KUKA KRL program: MyProgram_173().src

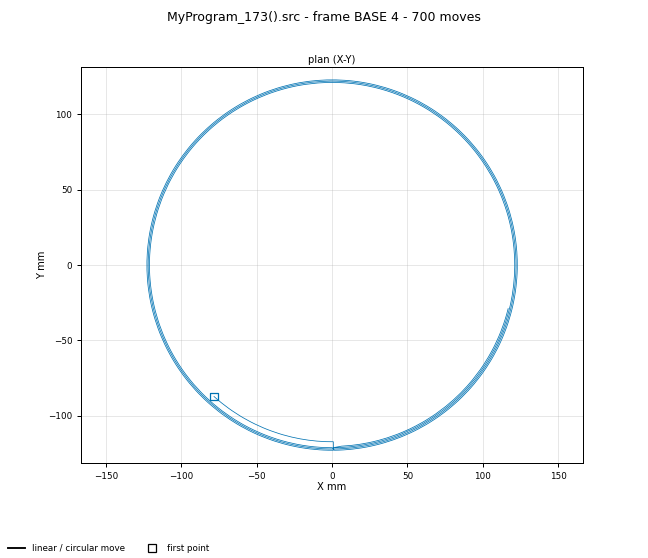
[picture p0: tool path of MyProgram_173().src in frame BASE 4, 700 of 700 moves have a stored position in this frame; points joined in program order, loops and branches not executed]
&ACCESS RVP
&REL 1
&PARAM TEMPLATE = C:\KRC\Roboter\Template\vorgabe
&PARAM EDITMASK = *
DEF MyProgram_173()
; ---- Setting reference (Base) ----
$BASE = BASE_DATA[4]

; --------------------------
; ---- Setting tool (TCP) ----
$TOOL = TOOL_DATA[3]
; --------------------------

$VEL.CP = VEL_APROX_PRINT
Startdeposition()
$VEL.CP = VEL_PRINT
LIN {X -78.3175,Y -87.2157,Z 128,A -135.2018,B 24.9548,C -1.5536,E1 24.894,E2 221.2459} C_DIS
LIN {X -76.0204,Y -89.2249,Z 128,A -133.7214,B 24.955,C -1.5502,E1 24.8972,E2 219.7678} C_DIS
LIN {X -73.3158,Y -91.4624,Z 128,A -132.0203,B 24.9552,C -1.5463,E1 24.9008,E2 218.0696} C_DIS
LIN {X -70.7779,Y -93.4392,Z 128,A -130.557,B 24.9556,C -1.5388,E1 24.904,E2 216.6188} C_DIS
LIN {X -68.6874,Y -94.988,Z 128,A -129.0705,B 24.9552,C -1.5458,E1 24.9074,E2 215.1104} C_DIS
LIN {X -66.3132,Y -96.6605,Z 128,A -127.7459,B 24.9556,C -1.5393,E1 24.9105,E2 213.7967} C_DIS
LIN {X -63.7074,Y -98.3959,Z 128,A -126.2103,B 24.9557,C -1.5371,E1 24.914,E2 212.2613} C_DIS
LIN {X -61.2786,Y -99.9267,Z 128,A -124.8024,B 24.9558,C -1.5352,E1 24.9174,E2 210.8536} C_DIS
LIN {X -58.8133,Y -101.3972,Z 128,A -123.3955,B 24.956,C -1.5333,E1 24.9208,E2 209.447} C_DIS
LIN {X -56.1243,Y -102.9093,Z 128,A -122.0747,B 24.9565,C -1.5231,E1 24.9239,E2 208.1466} C_DIS
LIN {X -53.9775,Y -104.0535,Z 128,A -120.6902,B 24.9561,C -1.53,E1 24.9274,E2 206.7418} C_DIS
LIN {X -51.181,Y -105.4557,Z 128,A -119.157,B 24.9562,C -1.5283,E1 24.9312,E2 205.2087} C_DIS
LIN {X -48.3648,Y -106.7758,Z 128,A -117.8498,B 24.9569,C -1.5172,E1 24.9345,E2 203.9245} C_DIS
LIN {X -45.8347,Y -107.8864,Z 128,A -116.3218,B 24.9565,C -1.5235,E1 24.9385,E2 202.378} C_DIS
LIN {X -43.5316,Y -108.8379,Z 128,A -114.9638,B 24.9562,C -1.5284,E1 24.942,E2 201.0053} C_DIS
LIN {X -40.5891,Y -109.9678,Z 128,A -113.5212,B 24.9566,C -1.5227,E1 24.9458,E2 199.5733} C_DIS
LIN {X -37.8192,Y -110.9506,Z 128,A -112.1239,B 24.9567,C -1.5197,E1 24.9494,E2 198.1804} C_DIS
LIN {X -35.2434,Y -111.7962,Z 128,A -110.8198,B 24.9568,C -1.5177,E1 24.9529,E2 196.8786} C_DIS
LIN {X -32.6052,Y -112.5946,Z 128,A -109.2722,B 24.9564,C -1.5257,E1 24.9571,E2 195.3097} C_DIS
LIN {X -29.336,Y -113.4884,Z 128,A -107.7138,B 24.9567,C -1.5203,E1 24.9613,E2 193.7616} C_DIS
LIN {X -26.8263,Y -114.1085,Z 128,A -106.5879,B 24.9571,C -1.5135,E1 24.9643,E2 192.6504} C_DIS
LIN {X -24.0235,Y -114.7313,Z 128,A -105.0697,B 24.9568,C -1.518,E1 24.9685,E2 191.1197} C_DIS
LIN {X -21.2072,Y -115.2851,Z 128,A -103.6628,B 24.9568,C -1.5176,E1 24.9723,E2 189.7121} C_DIS
LIN {X -18.6199,Y -115.7324,Z 128,A -102.2849,B 24.9566,C -1.5214,E1 24.9762,E2 188.3239} C_DIS
LIN {X -15.7808,Y -116.1536,Z 128,A -100.8781,B 24.9566,C -1.5213,E1 24.98,E2 186.9163} C_DIS
LIN {X -12.6612,Y -116.5336,Z 128,A -99.4416,B 24.9569,C -1.5166,E1 24.984,E2 185.49} C_DIS
LIN {X -10.0626,Y -116.788,Z 128,A -98.1635,B 24.9569,C -1.5166,E1 24.9876,E2 184.2113} C_DIS
LIN {X -6.9466,Y -117.0135,Z 128,A -96.6383,B 24.9569,C -1.5166,E1 24.9918,E2 182.6857} C_DIS
LIN {X -4.0837,Y -117.1484,Z 128,A -95.3376,B 24.9572,C -1.5121,E1 24.9954,E2 181.3951} C_DIS
LIN {X -1.1778,Y -117.2135,Z 128,A -93.9306,B 24.9572,C -1.5118,E1 24.9993,E2 179.9889} C_DIS
LIN {X 0.813,Y -117.2142,Z 128,A -93.1077,B 24.9576,C -1.5052,E1 25.0016,E2 179.1816} C_DIS
Enddeposition()
LIN {X 0.8728,Y -122.8508,Z 129,A -93.006,B 24.9623,C -1.4183,E1 25.0013,E2 179.2858} C_DIS
Startdeposition()
$VEL.CP = VEL_PRINT
LIN {X -2.5785,Y -122.8272,Z 129,A -94.9222,B 24.9631,C -1.4034,E1 24.9959,E2 181.2373} C_DIS
LIN {X -5.5921,Y -122.7269,Z 129,A -96.2871,B 24.9631,C -1.4052,E1 24.9921,E2 182.5982} C_DIS
LIN {X -8.6023,Y -122.5527,Z 129,A -97.6934,B 24.9631,C -1.4052,E1 24.9881,E2 184.0051} C_DIS
LIN {X -12.042,Y -122.2646,Z 129,A -99.303,B 24.9631,C -1.4052,E1 24.9837,E2 185.6154} C_DIS
LIN {X -14.6053,Y -121.983,Z 129,A -100.5473,B 24.9631,C -1.4035,E1 24.9802,E2 186.8646} C_DIS
LIN {X -17.5945,Y -121.5879,Z 129,A -101.9132,B 24.963,C -1.4057,E1 24.9764,E2 188.2263} C_DIS
LIN {X -20.5731,Y -121.1195,Z 129,A -103.3204,B 24.963,C -1.4061,E1 24.9725,E2 189.634} C_DIS
LIN {X -23.5393,Y -120.5781,Z 129,A -104.7183,B 24.963,C -1.407,E1 24.9687,E2 191.0311} C_DIS
LIN {X -26.9179,Y -119.871,Z 129,A -106.339,B 24.963,C -1.4072,E1 24.9643,E2 192.6533} C_DIS
LIN {X -29.8516,Y -119.1743,Z 129,A -107.7472,B 24.9629,C -1.4079,E1 24.9605,E2 194.0619} C_DIS
LIN {X -32.7673,Y -118.4058,Z 129,A -109.155,B 24.9629,C -1.4087,E1 24.9567,E2 195.4699} C_DIS
LIN {X -35.6633,Y -117.566,Z 129,A -110.5633,B 24.9628,C -1.4096,E1 24.9529,E2 196.8785} C_DIS
LIN {X -38.1224,Y -116.7898,Z 129,A -111.7683,B 24.9628,C -1.4104,E1 24.9497,E2 198.0836} C_DIS
LIN {X -41.389,Y -115.6745,Z 129,A -113.3811,B 24.9627,C -1.4117,E1 24.9454,E2 199.6966} C_DIS
LIN {X -44.0204,Y -114.6977,Z 129,A -114.7031,B 24.9627,C -1.4123,E1 24.942,E2 201.0198} C_DIS
LIN {X -46.6107,Y -113.6689,Z 129,A -116.0365,B 24.9627,C -1.4121,E1 24.9385,E2 202.3567} C_DIS
LIN {X -49.3862,Y -112.4908,Z 129,A -117.4048,B 24.9625,C -1.4154,E1 24.935,E2 203.7205} C_DIS
LIN {X -52.5278,Y -111.0607,Z 129,A -119.0187,B 24.9624,C -1.417,E1 24.9309,E2 205.3344} C_DIS
LIN {X -55.2375,Y -109.7381,Z 129,A -120.4286,B 24.9624,C -1.4186,E1 24.9274,E2 206.7443} C_DIS
LIN {X -57.914,Y -108.3495,Z 129,A -121.8387,B 24.9622,C -1.4203,E1 24.9239,E2 208.1543} C_DIS
LIN {X -60.1744,Y -107.1084,Z 129,A -123.0452,B 24.9622,C -1.4218,E1 24.921,E2 209.3606} C_DIS
LIN {X -63.1607,Y -105.3773,Z 129,A -124.6598,B 24.962,C -1.4239,E1 24.9171,E2 210.9751} C_DIS
LIN {X -65.7278,Y -103.7955,Z 129,A -126.0709,B 24.962,C -1.4259,E1 24.9137,E2 212.386} C_DIS
LIN {X -67.8803,Y -102.3984,Z 129,A -127.3153,B 24.962,C -1.4256,E1 24.9108,E2 213.635} C_DIS
LIN {X -70.7416,Y -100.4453,Z 129,A -128.8932,B 24.9617,C -1.43,E1 24.9072,E2 215.2078} C_DIS
LIN {X -72.8331,Y -98.9369,Z 129,A -130.1005,B 24.9616,C -1.4319,E1 24.9045,E2 216.4148} C_DIS
LIN {X -75.2392,Y -97.1197,Z 129,A -131.5534,B 24.9616,C -1.4324,E1 24.9013,E2 217.8719} C_DIS
LIN {X -77.9391,Y -94.9691,Z 129,A -133.1283,B 24.9613,C -1.4369,E1 24.8979,E2 219.4419} C_DIS
LIN {X -79.914,Y -93.3109,Z 129,A -134.336,B 24.9613,C -1.4391,E1 24.8953,E2 220.6492} C_DIS
LIN {X -82.1799,Y -91.3216,Z 129,A -135.7483,B 24.9611,C -1.4416,E1 24.8923,E2 222.061} C_DIS
LIN {X -84.7143,Y -88.9782,Z 129,A -137.3655,B 24.9609,C -1.4446,E1 24.889,E2 223.6778} C_DIS
LIN {X -86.8724,Y -86.8724,Z 129,A -138.7777,B 24.9608,C -1.4473,E1 24.8862,E2 225.0895} C_DIS
LIN {X -88.6753,Y -85.0287,Z 129,A -139.9861,B 24.9606,C -1.4498,E1 24.8839,E2 226.2973} C_DIS
LIN {X -90.7691,Y -82.79,Z 129,A -141.4561,B 24.9606,C -1.4512,E1 24.8811,E2 227.7704} C_DIS
LIN {X -93.0278,Y -80.2463,Z 129,A -143.017,B 24.9603,C -1.4559,E1 24.8782,E2 229.3269} C_DIS
LIN {X -94.6901,Y -78.2749,Z 129,A -144.2259,B 24.9601,C -1.4585,E1 24.8761,E2 230.5353} C_DIS
LIN {X -96.5825,Y -75.9275,Z 129,A -145.6807,B 24.9601,C -1.4598,E1 24.8735,E2 231.994} C_DIS
LIN {X -98.679,Y -73.1853,Z 129,A -147.2578,B 24.9598,C -1.4652,E1 24.8709,E2 233.5657} C_DIS
LIN {X -100.4453,Y -70.7416,Z 129,A -148.6716,B 24.9596,C -1.4684,E1 24.8686,E2 234.9787} C_DIS
LIN {X -101.9064,Y -68.6167,Z 129,A -149.881,B 24.9594,C -1.4712,E1 24.8667,E2 236.1874} C_DIS
LIN {X -103.5597,Y -66.0952,Z 129,A -151.2749,B 24.9592,C -1.4755,E1 24.8646,E2 237.5782} C_DIS
LIN {X -105.1505,Y -63.5338,Z 129,A -152.7094,B 24.9591,C -1.478,E1 24.8625,E2 239.0141} C_DIS
LIN {X -106.8956,Y -60.5556,Z 129,A -154.3286,B 24.9589,C -1.4819,E1 24.8602,E2 240.6324} C_DIS
LIN {X -108.3495,Y -57.914,Z 129,A -155.7433,B 24.9587,C -1.4854,E1 24.8583,E2 242.0461} C_DIS
LIN {X -109.5394,Y -55.6263,Z 129,A -156.9533,B 24.9585,C -1.4885,E1 24.8568,E2 243.2553} C_DIS
LIN {X -111.0607,Y -52.5278,Z 129,A -158.5729,B 24.9583,C -1.4927,E1 24.8548,E2 244.8738} C_DIS
LIN {X -112.3163,Y -49.7864,Z 129,A -159.9877,B 24.9581,C -1.4963,E1 24.8532,E2 246.2876} C_DIS
LIN {X -113.3348,Y -47.4173,Z 129,A -161.2395,B 24.958,C -1.4977,E1 24.8519,E2 247.543} C_DIS
LIN {X -114.4643,Y -44.6217,Z 129,A -162.6133,B 24.9577,C -1.5033,E1 24.8504,E2 248.9112} C_DIS
LIN {X -115.5249,Y -41.7991,Z 129,A -164.0285,B 24.9574,C -1.5071,E1 24.8491,E2 250.3253} C_DIS
LIN {X -116.6554,Y -38.5377,Z 129,A -165.6487,B 24.9572,C -1.5115,E1 24.8476,E2 251.9443} C_DIS
LIN {X -117.4367,Y -36.0803,Z 129,A -166.8595,B 24.957,C -1.5149,E1 24.8466,E2 253.154} C_DIS
LIN {X -118.2868,Y -33.1874,Z 129,A -168.275,B 24.9568,C -1.5188,E1 24.8455,E2 254.5683} C_DIS
LIN {X -119.0657,Y -30.2745,Z 129,A -169.6906,B 24.9566,C -1.5228,E1 24.8445,E2 255.9828} C_DIS
LIN {X -119.801,Y -27.2211,Z 129,A -171.1534,B 24.9563,C -1.5274,E1 24.8436,E2 257.443} C_DIS
LIN {X -120.4955,Y -23.9681,Z 129,A -172.727,B 24.9561,C -1.5313,E1 24.8427,E2 259.0166} C_DIS
LIN {X -121.0193,Y -21.1602,Z 129,A -174.0531,B 24.9558,C -1.5358,E1 24.842,E2 260.3399} C_DIS
LIN {X -121.5265,Y -18.0267,Z 129,A -175.5587,B 24.9556,C -1.5395,E1 24.8414,E2 261.8458} C_DIS
LIN {X -121.8761,Y -15.4719,Z 129,A -176.8112,B 24.9555,C -1.5412,E1 24.8409,E2 263.1016} C_DIS
LIN {X -122.2191,Y -12.4762,Z 129,A -178.1858,B 24.9552,C -1.5471,E1 24.8405,E2 264.4704} C_DIS
LIN {X -122.5233,Y -9.0379,Z 129,A -179.807,B 24.9549,C -1.5518,E1 24.8402,E2 266.0901} C_DIS
LIN {X -122.7082,Y -6.0283,Z 129,A 178.7771,B 24.9546,C -1.5559,E1 24.8399,E2 267.5046} C_DIS
LIN {X -122.8058,Y -3.4514,Z 129,A 177.5245,B 24.9546,C -1.5577,E1 24.8399,E2 268.7605} C_DIS
LIN {X -122.8542,Y -0.3629,Z 129,A 176.0949,B 24.9542,C -1.5629,E1 24.8398,E2 270.1864} C_DIS
LIN {X -122.8272,Y 2.5785,Z 129,A 174.6923,B 24.954,C -1.5661,E1 24.8398,E2 271.5899} C_DIS
LIN {X -122.7269,Y 5.5921,Z 129,A 173.3176,B 24.9537,C -1.572,E1 24.84,E2 272.9587} C_DIS
LIN {X -122.5604,Y 8.4883,Z 129,A 171.9386,B 24.9535,C -1.5753,E1 24.8402,E2 274.3381} C_DIS
LIN {X -122.2646,Y 12.042,Z 129,A 170.2806,B 24.9532,C -1.581,E1 24.8407,E2 275.9927} C_DIS
LIN {X -121.9322,Y 15.0389,Z 129,A 168.8642,B 24.9529,C -1.5851,E1 24.8411,E2 277.4076} C_DIS
LIN {X -121.5879,Y 17.5945,Z 129,A 167.6531,B 24.9527,C -1.5887,E1 24.8416,E2 278.6174} C_DIS
LIN {X -121.0475,Y 21.0037,Z 129,A 166.0319,B 24.9524,C -1.5934,E1 24.8423,E2 280.237} C_DIS
LIN {X -120.4955,Y 23.9681,Z 129,A 164.616,B 24.9522,C -1.5976,E1 24.8431,E2 281.6513} C_DIS
LIN {X -119.871,Y 26.9179,Z 129,A 163.2,B 24.9519,C -1.6017,E1 24.8439,E2 283.0658} C_DIS
LIN {X -119.1743,Y 29.8516,Z 129,A 161.7838,B 24.9517,C -1.6058,E1 24.8448,E2 284.4805} C_DIS
LIN {X -118.4058,Y 32.7673,Z 129,A 160.368,B 24.9514,C -1.6099,E1 24.8459,E2 285.8947} C_DIS
LIN {X -117.566,Y 35.6633,Z 129,A 158.9522,B 24.9512,C -1.614,E1 24.847,E2 287.3091} C_DIS
LIN {X -116.6554,Y 38.5377,Z 129,A 157.5361,B 24.9509,C -1.618,E1 24.8482,E2 288.7237} C_DIS
LIN {X -115.8191,Y 40.977,Z 129,A 156.3254,B 24.9507,C -1.6215,E1 24.8493,E2 289.9329} C_DIS
LIN {X -114.7786,Y 43.807,Z 129,A 154.8682,B 24.9506,C -1.6237,E1 24.8507,E2 291.3931} C_DIS
LIN {X -113.6689,Y 46.6107,Z 129,A 153.4526,B 24.9504,C -1.6277,E1 24.8522,E2 292.8072} C_DIS
LIN {X -112.4908,Y 49.3862,Z 129,A 152.0784,B 24.95,C -1.6334,E1 24.8537,E2 294.1753} C_DIS
LIN {X -111.0607,Y 52.5278,Z 129,A 150.4581,B 24.9497,C -1.6378,E1 24.8556,E2 295.794} C_DIS
LIN {X -109.932,Y 54.8464,Z 129,A 149.2062,B 24.9497,C -1.6393,E1 24.8572,E2 297.0489} C_DIS
LIN {X -108.3495,Y 57.914,Z 129,A 147.6276,B 24.9493,C -1.6455,E1 24.8592,E2 298.6213} C_DIS
LIN {X -107.1084,Y 60.1744,Z 129,A 146.3944,B 24.9491,C -1.6477,E1 24.8609,E2 299.8556} C_DIS
LIN {X -105.3773,Y 63.1607,Z 129,A 144.7972,B 24.9488,C -1.6529,E1 24.8632,E2 301.4487} C_DIS
LIN {X -103.7955,Y 65.7278,Z 129,A 143.3822,B 24.9486,C -1.6566,E1 24.8652,E2 302.8621} C_DIS
LIN {X -102.1512,Y 68.2552,Z 129,A 141.9675,B 24.9483,C -1.6602,E1 24.8674,E2 304.2753} C_DIS
LIN {X -100.4454,Y 70.7416,Z 129,A 140.5528,B 24.9481,C -1.6638,E1 24.8697,E2 305.6885} C_DIS
LIN {X -98.9369,Y 72.8331,Z 129,A 139.3428,B 24.9479,C -1.6668,E1 24.8717,E2 306.8971} C_DIS
LIN {X -97.1197,Y 75.2392,Z 129,A 137.9283,B 24.9477,C -1.6703,E1 24.8741,E2 308.3102} C_DIS
LIN {X -95.2749,Y 77.5618,Z 129,A 136.5307,B 24.9475,C -1.6734,E1 24.8765,E2 309.7069} C_DIS
LIN {X -93.3109,Y 79.914,Z 129,A 135.0585,B 24.9475,C -1.6752,E1 24.8792,E2 311.1814} C_DIS
LIN {X -91.0304,Y 82.5052,Z 129,A 133.4814,B 24.9471,C -1.6808,E1 24.8821,E2 312.7524} C_DIS
LIN {X -88.9782,Y 84.7143,Z 129,A 132.0672,B 24.9469,C -1.684,E1 24.8848,E2 314.1652} C_DIS
LIN {X -86.8724,Y 86.8724,Z 129,A 130.6539,B 24.9467,C -1.6871,E1 24.8875,E2 315.577} C_DIS
LIN {X -84.7143,Y 88.9782,Z 129,A 129.2402,B 24.9465,C -1.6902,E1 24.8904,E2 316.9893} C_DIS
LIN {X -82.6505,Y 90.8971,Z 129,A 127.9097,B 24.9463,C -1.6926,E1 24.8931,E2 318.3195} C_DIS
LIN {X -80.5751,Y 92.7406,Z 129,A 126.6269,B 24.9461,C -1.6961,E1 24.8958,E2 319.5989} C_DIS
LIN {X -78.2749,Y 94.6901,Z 129,A 125.2051,B 24.9459,C -1.6986,E1 24.8988,E2 321.0203} C_DIS
LIN {X -75.9275,Y 96.5825,Z 129,A 123.7923,B 24.9458,C -1.7014,E1 24.9019,E2 322.4317} C_DIS
LIN {X -73.5344,Y 98.4168,Z 129,A 122.3381,B 24.9457,C -1.7022,E1 24.9052,E2 323.8891} C_DIS
LIN {X -71.1398,Y 100.1613,Z 129,A 120.9848,B 24.9454,C -1.7064,E1 24.9082,E2 325.2373} C_DIS
LIN {X -68.6167,Y 101.9064,Z 129,A 119.5548,B 24.9452,C -1.7093,E1 24.9115,E2 326.6652} C_DIS
LIN {X -66.0952,Y 103.5597,Z 129,A 118.1429,B 24.9451,C -1.7117,E1 24.9148,E2 328.0758} C_DIS
LIN {X -63.5338,Y 105.1505,Z 129,A 116.7309,B 24.9449,C -1.7141,E1 24.9182,E2 329.4866} C_DIS
LIN {X -60.5556,Y 106.8956,Z 129,A 115.1146,B 24.9448,C -1.7167,E1 24.9221,E2 331.1015} C_DIS
LIN {X -57.914,Y 108.3495,Z 129,A 113.7034,B 24.9446,C -1.7189,E1 24.9256,E2 332.5115} C_DIS
LIN {X -55.4274,Y 109.6411,Z 129,A 112.4075,B 24.9445,C -1.7216,E1 24.9288,E2 333.8045} C_DIS
LIN {X -52.5278,Y 111.0607,Z 129,A 110.881,B 24.9444,C -1.723,E1 24.9326,E2 335.3314} C_DIS
LIN {X -49.7864,Y 112.3163,Z 129,A 109.4703,B 24.9442,C -1.725,E1 24.9362,E2 336.741} C_DIS
LIN {X -47.4173,Y 113.3348,Z 129,A 108.2224,B 24.9442,C -1.7247,E1 24.9394,E2 337.9923} C_DIS
LIN {X -44.6217,Y 114.4643,Z 129,A 106.8532,B 24.944,C -1.7283,E1 24.943,E2 339.3559} C_DIS
LIN {X -41.7991,Y 115.5249,Z 129,A 105.4431,B 24.944,C -1.73,E1 24.9466,E2 340.765} C_DIS
LIN {X -38.5377,Y 116.6554,Z 129,A 103.8291,B 24.9438,C -1.7318,E1 24.9509,E2 342.3778} C_DIS
LIN {X -36.0803,Y 117.4367,Z 129,A 102.6232,B 24.9438,C -1.7331,E1 24.9541,E2 343.5827} C_DIS
LIN {X -33.1874,Y 118.2868,Z 129,A 101.1725,B 24.9438,C -1.7326,E1 24.958,E2 345.037} C_DIS
LIN {X -29.8516,Y 119.1743,Z 129,A 99.6006,B 24.9435,C -1.7359,E1 24.9623,E2 346.6034} C_DIS
LIN {X -27.296,Y 119.7837,Z 129,A 98.378,B 24.9435,C -1.7372,E1 24.9656,E2 347.8245} C_DIS
LIN {X -23.9681,Y 120.4955,Z 129,A 96.7827,B 24.9434,C -1.7381,E1 24.9699,E2 349.4194} C_DIS
LIN {X -21.0037,Y 121.0475,Z 129,A 95.3741,B 24.9434,C -1.7391,E1 24.9738,E2 350.8271} C_DIS
LIN {X -18.0267,Y 121.5265,Z 129,A 93.9659,B 24.9433,C -1.74,E1 24.9777,E2 352.2345} C_DIS
LIN {X -15.4719,Y 121.8761,Z 129,A 92.7616,B 24.9433,C -1.7407,E1 24.981,E2 353.438} C_DIS
LIN {X -12.042,Y 122.2646,Z 129,A 91.1499,B 24.9432,C -1.7415,E1 24.9855,E2 355.0489} C_DIS
LIN {X -9.4731,Y 122.4885,Z 129,A 89.9457,B 24.9432,C -1.742,E1 24.9888,E2 356.2523} C_DIS
LIN {X -6.0283,Y 122.7082,Z 129,A 88.3348,B 24.9431,C -1.7425,E1 24.9933,E2 357.8625} C_DIS
LIN {X -3.5053,Y 122.8041,Z 129,A 87.1059,B 24.9432,C -1.7405,E1 24.9968,E2 359.0963} C_DIS
LIN {X 0,Y 122.8562,Z 129,A 85.5207,B 24.9431,C -1.7432,E1 25.0012,E2 360.6753} C_DIS
LIN {X 2.5785,Y 122.8272,Z 129,A 84.2766,B 24.9431,C -1.7414,E1 25.0047,E2 361.9233} C_DIS
LIN {X 5.5921,Y 122.7269,Z 129,A 82.9112,B 24.9431,C -1.7434,E1 25.0085,E2 363.2836} C_DIS
LIN {X 8.5036,Y 122.5594,Z 129,A 81.5373,B 24.9431,C -1.7428,E1 25.0123,E2 364.6585} C_DIS
LIN {X 11.6073,Y 122.3047,Z 129,A 80.0581,B 24.9431,C -1.7414,E1 25.0164,E2 366.1401} C_DIS
LIN {X 14.6053,Y 121.983,Z 129,A 78.6935,B 24.9431,C -1.7431,E1 25.0202,E2 367.4998} C_DIS
LIN {X 17.5945,Y 121.5879,Z 129,A 77.247,B 24.9432,C -1.7408,E1 25.0242,E2 368.9503} C_DIS
LIN {X 20.5731,Y 121.1195,Z 129,A 75.8414,B 24.9432,C -1.7404,E1 25.0281,E2 370.3555} C_DIS
LIN {X 23.8641,Y 120.5155,Z 129,A 74.3206,B 24.9432,C -1.7416,E1 25.0322,E2 371.8717} C_DIS
LIN {X 26.9179,Y 119.871,Z 129,A 72.8697,B 24.9432,C -1.7411,E1 25.0362,E2 373.322} C_DIS
LIN {X 29.8516,Y 119.1743,Z 129,A 71.465,B 24.9432,C -1.7403,E1 25.04,E2 374.7265} C_DIS
LIN {X 32.7673,Y 118.4058,Z 129,A 70.0609,B 24.9432,C -1.7395,E1 25.0438,E2 376.1303} C_DIS
LIN {X 35.1793,Y 117.7096,Z 129,A 68.8387,B 24.9435,C -1.7362,E1 25.0471,E2 377.358} C_DIS
LIN {X 38.1224,Y 116.7898,Z 129,A 67.4561,B 24.9435,C -1.7377,E1 25.0507,E2 378.7347} C_DIS
LIN {X 40.977,Y 115.8191,Z 129,A 66.0524,B 24.9435,C -1.7366,E1 25.0544,E2 380.1382} C_DIS
LIN {X 43.8071,Y 114.7786,Z 129,A 64.6082,B 24.9437,C -1.7334,E1 25.0582,E2 381.5868} C_DIS
LIN {X 46.6107,Y 113.6689,Z 129,A 63.205,B 24.9437,C -1.7321,E1 25.0619,E2 382.9899} C_DIS
LIN {X 49.7864,Y 112.3163,Z 129,A 61.6401,B 24.9437,C -1.7324,E1 25.0659,E2 384.5503} C_DIS
LIN {X 52.132,Y 111.2449,Z 129,A 60.3993,B 24.944,C -1.7292,E1 25.069,E2 385.7956} C_DIS
LIN {X 55.2375,Y 109.7381,Z 129,A 58.8351,B 24.944,C -1.7292,E1 25.0729,E2 387.3554} C_DIS
LIN {X 57.914,Y 108.3495,Z 129,A 57.4328,B 24.944,C -1.7275,E1 25.0764,E2 388.7578} C_DIS
LIN {X 60.5556,Y 106.8956,Z 129,A 56.0307,B 24.9442,C -1.7257,E1 25.0798,E2 390.16} C_DIS
LIN {X 62.7849,Y 105.5994,Z 129,A 54.791,B 24.9444,C -1.7222,E1 25.0828,E2 391.4043} C_DIS
LIN {X 65.7278,Y 103.7955,Z 129,A 53.2273,B 24.9444,C -1.7219,E1 25.0865,E2 392.9637} C_DIS
LIN {X 68.2552,Y 102.1512,Z 129,A 51.826,B 24.9446,C -1.7198,E1 25.0898,E2 394.3654} C_DIS
LIN {X 70.7416,Y 100.4453,Z 129,A 50.425,B 24.9447,C -1.7177,E1 25.093,E2 395.7666} C_DIS
LIN {X 72.8331,Y 98.9369,Z 129,A 49.2269,B 24.9448,C -1.7158,E1 25.0957,E2 396.9649} C_DIS
LIN {X 75.585,Y 96.8532,Z 129,A 47.6233,B 24.945,C -1.7131,E1 25.0992,E2 398.5689} C_DIS
LIN {X 77.9391,Y 94.9691,Z 129,A 46.2225,B 24.9452,C -1.7107,E1 25.1023,E2 399.9701} C_DIS
LIN {X 79.9908,Y 93.2455,Z 129,A 44.9527,B 24.9454,C -1.7073,E1 25.105,E2 401.2431} C_DIS
LIN {X 82.1155,Y 91.3793,Z 129,A 43.6531,B 24.9454,C -1.7056,E1 25.1077,E2 402.5416} C_DIS
LIN {X 84.3963,Y 89.2773,Z 129,A 42.1839,B 24.9457,C -1.7015,E1 25.1107,E2 404.0145} C_DIS
LIN {X 87.6251,Y 86.1104,Z 129,A 40.1252,B 24.9459,C -1.6994,E1 25.1148,E2 406.0694} C_DIS
LIN {X 89.712,Y 83.9341,Z 129,A 38.7256,B 24.9461,C -1.6966,E1 25.1175,E2 407.4696} C_DIS
LIN {X 91.7448,Y 81.7071,Z 129,A 37.326,B 24.9462,C -1.6937,E1 25.1201,E2 408.8698} C_DIS
LIN {X 93.7961,Y 79.3445,Z 129,A 35.8504,B 24.9465,C -1.6894,E1 25.1228,E2 410.3488} C_DIS
LIN {X 95.6435,Y 77.107,Z 129,A 34.4869,B 24.9468,C -1.6856,E1 25.1252,E2 411.7148} C_DIS
LIN {X 97.7735,Y 74.3908,Z 129,A 32.9266,B 24.9468,C -1.6841,E1 25.1279,E2 413.2714} C_DIS
LIN {X 99.5697,Y 71.9689,Z 129,A 31.5278,B 24.9471,C -1.6809,E1 25.1302,E2 414.671} C_DIS
LIN {X 101.3059,Y 69.5036,Z 129,A 30.129,B 24.9473,C -1.6777,E1 25.1324,E2 416.0705} C_DIS
LIN {X 102.9811,Y 66.9965,Z 129,A 28.7305,B 24.9475,C -1.6744,E1 25.1345,E2 417.4699} C_DIS
LIN {X 104.5943,Y 64.4491,Z 129,A 27.3326,B 24.9477,C -1.671,E1 25.1366,E2 418.8686} C_DIS
LIN {X 106.1444,Y 61.8628,Z 129,A 25.9345,B 24.9479,C -1.6676,E1 25.1386,E2 420.2676} C_DIS
LIN {X 107.5988,Y 59.2962,Z 129,A 24.5754,B 24.9481,C -1.6646,E1 25.1405,E2 421.6266} C_DIS
LIN {X 109.052,Y 56.58,Z 129,A 23.1384,B 24.9483,C -1.6606,E1 25.1423,E2 423.0655} C_DIS
LIN {X 110.4077,Y 53.8867,Z 129,A 21.7407,B 24.9485,C -1.657,E1 25.1441,E2 424.4642} C_DIS
LIN {X 111.5127,Y 51.5567,Z 129,A 20.5614,B 24.9487,C -1.6548,E1 25.1455,E2 425.6424} C_DIS
LIN {X 112.7444,Y 48.8046,Z 129,A 19.1477,B 24.949,C -1.6503,E1 25.1471,E2 427.059} C_DIS
LIN {X 113.9081,Y 46.023,Z 129,A 17.7502,B 24.9492,C -1.6466,E1 25.1485,E2 428.4576} C_DIS
LIN {X 115.1579,Y 42.8054,Z 129,A 16.1505,B 24.9495,C -1.6422,E1 25.1501,E2 430.0586} C_DIS
LIN {X 116.0292,Y 40.3783,Z 129,A 14.9558,B 24.9497,C -1.639,E1 25.1512,E2 431.2541} C_DIS
LIN {X 116.9851,Y 37.5187,Z 129,A 13.5584,B 24.9499,C -1.6352,E1 25.1525,E2 432.6526} C_DIS
LIN {X 117.8707,Y 34.6364,Z 129,A 12.1774,B 24.9501,C -1.6321,E1 25.1536,E2 434.033} C_DIS
LIN {X 118.799,Y 31.3118,Z 129,A 10.5624,B 24.9504,C -1.6269,E1 25.1548,E2 435.6512} C_DIS
LIN {X 119.4062,Y 28.9012,Z 129,A 9.3531,B 24.9508,C -1.6208,E1 25.1556,E2 436.8679} C_DIS
LIN {X 120.1583,Y 25.6011,Z 129,A 7.836,B 24.9508,C -1.6188,E1 25.1565,E2 438.3807} C_DIS
LIN {X 120.7806,Y 22.4876,Z 129,A 6.3718,B 24.9511,C -1.615,E1 25.1573,E2 439.8455} C_DIS
LIN {X 121.2961,Y 19.5167,Z 129,A 4.9748,B 24.9514,C -1.6109,E1 25.1579,E2 441.2437} C_DIS
LIN {X 121.7385,Y 16.5341,Z 129,A 3.5783,B 24.9516,C -1.6069,E1 25.1585,E2 442.6416} C_DIS
LIN {X 122.1076,Y 13.5415,Z 129,A 2.1817,B 24.9519,C -1.6028,E1 25.1589,E2 444.0395} C_DIS
LIN {X 122.5233,Y 9.0379,Z 129,A 0.0866,B 24.9522,C -1.5967,E1 25.1594,E2 446.1365} C_DIS
LIN {X 122.7082,Y 6.0283,Z 129,A -1.3098,B 24.9525,C -1.5926,E1 25.1596,E2 447.5343} C_DIS
LIN {X 122.8058,Y 3.4514,Z 129,A -2.5451,B 24.9528,C -1.5871,E1 25.1597,E2 448.7753} C_DIS
LIN {X 122.8542,Y 0.3629,Z 129,A -3.9703,B 24.953,C -1.5831,E1 25.1597,E2 450.2014} C_DIS
LIN {X 122.8272,Y -2.5785,Z 129,A -5.338,B 24.9533,C -1.5788,E1 25.1597,E2 451.571} C_DIS
LIN {X 122.7269,Y -5.5921,Z 129,A -6.6937,B 24.9534,C -1.5768,E1 25.1596,E2 452.9235} C_DIS
LIN {X 122.5527,Y -8.6023,Z 129,A -8.0902,B 24.9537,C -1.5726,E1 25.1593,E2 454.3215} C_DIS
LIN {X 122.2999,Y -11.6591,Z 129,A -9.5431,B 24.954,C -1.5668,E1 25.159,E2 455.7795} C_DIS
LIN {X 121.983,Y -14.6053,Z 129,A -10.9238,B 24.9543,C -1.5623,E1 25.1585,E2 457.1626} C_DIS
LIN {X 121.5879,Y -17.5945,Z 129,A -12.2795,B 24.9543,C -1.5603,E1 25.158,E2 458.5152} C_DIS
LIN {X 121.1195,Y -20.5731,Z 129,A -13.6761,B 24.9546,C -1.5562,E1 25.1574,E2 459.9133} C_DIS
LIN {X 120.5781,Y -23.5393,Z 129,A -15.0726,B 24.9549,C -1.5521,E1 25.1567,E2 461.3113} C_DIS
LIN {X 119.871,Y -26.9179,Z 129,A -16.6712,B 24.9551,C -1.5474,E1 25.1557,E2 462.9116} C_DIS
LIN {X 119.1743,Y -29.8516,Z 129,A -18.0681,B 24.9554,C -1.5433,E1 25.1548,E2 464.31} C_DIS
LIN {X 118.4058,Y -32.7673,Z 129,A -19.4644,B 24.9556,C -1.5393,E1 25.1538,E2 465.7078} C_DIS
LIN {X 117.566,Y -35.6633,Z 129,A -20.8611,B 24.9558,C -1.5352,E1 25.1527,E2 467.106} C_DIS
LIN {X 116.7898,Y -38.1224,Z 129,A -22.056,B 24.956,C -1.5318,E1 25.1516,E2 468.3021} C_DIS
LIN {X 115.6745,Y -41.389,Z 129,A -23.655,B 24.9563,C -1.5272,E1 25.1502,E2 469.903} C_DIS
LIN {X 114.6239,Y -44.2153,Z 129,A -25.0516,B 24.9565,C -1.5233,E1 25.1488,E2 471.301} C_DIS
LIN {X 113.6689,Y -46.6107,Z 129,A -26.2873,B 24.9568,C -1.5179,E1 25.1475,E2 472.5426} C_DIS
LIN {X 112.4908,Y -49.3862,Z 129,A -27.6435,B 24.9569,C -1.5161,E1 25.146,E2 473.8958} C_DIS
LIN {X 111.1786,Y -52.2744,Z 129,A -29.0999,B 24.9571,C -1.5127,E1 25.1443,E2 475.3523} C_DIS
LIN {X 109.7381,Y -55.2375,Z 129,A -30.64,B 24.9574,C -1.5078,E1 25.1424,E2 476.8956} C_DIS
LIN {X 108.3495,Y -57.914,Z 129,A -32.0372,B 24.9576,C -1.504,E1 25.1406,E2 478.2944} C_DIS
LIN {X 107.1084,Y -60.1744,Z 129,A -33.2325,B 24.9578,C -1.5009,E1 25.1389,E2 479.4909} C_DIS
LIN {X 105.3773,Y -63.1607,Z 129,A -34.8321,B 24.958,C -1.4966,E1 25.1367,E2 481.0923} C_DIS
LIN {X 103.7955,Y -65.7278,Z 129,A -36.2299,B 24.9582,C -1.493,E1 25.1346,E2 482.4916} C_DIS
LIN {X 102.3281,Y -67.9869,Z 129,A -37.5022,B 24.9585,C -1.4886,E1 25.1326,E2 483.7679} C_DIS
LIN {X 99.8389,Y -71.5916,Z 129,A -39.5128,B 24.9587,C -1.4845,E1 25.1294,E2 485.7784} C_DIS
LIN {X 98.0357,Y -74.0417,Z 129,A -40.92,B 24.9589,C -1.4811,E1 25.1271,E2 487.1867} C_DIS
LIN {X 95.9987,Y -76.6663,Z 129,A -42.4648,B 24.9591,C -1.4771,E1 25.1244,E2 488.7337} C_DIS
LIN {X 94.3423,Y -78.6934,Z 129,A -43.687,B 24.9593,C -1.4738,E1 25.1222,E2 489.9581} C_DIS
LIN {X 92.3232,Y -81.053,Z 129,A -45.1149,B 24.9595,C -1.471,E1 25.1196,E2 491.3861} C_DIS
LIN {X 90.3063,Y -83.2944,Z 129,A -46.5543,B 24.9598,C -1.4658,E1 25.1169,E2 492.8316} C_DIS
LIN {X 88.2097,Y -85.5116,Z 129,A -47.9641,B 24.9599,C -1.4628,E1 25.1142,E2 494.2422} C_DIS
LIN {X 86.1104,Y -87.6251,Z 129,A -49.3111,B 24.9599,C -1.4615,E1 25.1115,E2 495.5867} C_DIS
LIN {X 83.9341,Y -89.712,Z 129,A -50.7509,B 24.9603,C -1.4564,E1 25.1086,E2 497.0325} C_DIS
LIN {X 81.3819,Y -92.036,Z 129,A -52.3118,B 24.9603,C -1.455,E1 25.1053,E2 498.5904} C_DIS
LIN {X 79.0987,Y -94.0055,Z 129,A -53.7112,B 24.9605,C -1.4521,E1 25.1024,E2 499.9912} C_DIS
LIN {X 77.107,Y -95.6435,Z 129,A -54.9081,B 24.9606,C -1.4497,E1 25.0998,E2 501.1892} C_DIS
LIN {X 74.3908,Y -97.7735,Z 129,A -56.5105,B 24.9608,C -1.4466,E1 25.0962,E2 502.7932} C_DIS
LIN {X 71.9689,Y -99.5697,Z 129,A -57.9104,B 24.9609,C -1.4439,E1 25.0931,E2 504.1945} C_DIS
LIN {X 69.8621,Y -101.0567,Z 129,A -59.1078,B 24.9611,C -1.4417,E1 25.0903,E2 505.393} C_DIS
LIN {X 67.5077,Y -102.644,Z 129,A -60.4533,B 24.9613,C -1.438,E1 25.0872,E2 506.7427} C_DIS
LIN {X 64.8194,Y -104.363,Z 129,A -61.9087,B 24.9613,C -1.4367,E1 25.0838,E2 508.1965} C_DIS
LIN {X 62.2386,Y -105.9223,Z 129,A -63.3501,B 24.9616,C -1.4323,E1 25.0803,E2 509.6437} C_DIS
LIN {X 59.4374,Y -107.52,Z 129,A -64.8198,B 24.9616,C -1.4313,E1 25.0767,E2 511.1117} C_DIS
LIN {X 56.9663,Y -108.8486,Z 129,A -66.111,B 24.9617,C -1.4299,E1 25.0735,E2 512.4025} C_DIS
LIN {X 54.2779,Y -110.2138,Z 129,A -67.5532,B 24.9619,C -1.4258,E1 25.0699,E2 513.8505} C_DIS
LIN {X 51.5567,Y -111.5127,Z 129,A -68.9548,B 24.962,C -1.4237,E1 25.0664,E2 515.2533} C_DIS
LIN {X 48.4044,Y -112.9188,Z 129,A -70.5184,B 24.962,C -1.4235,E1 25.0624,E2 516.8136} C_DIS
LIN {X 45.9083,Y -113.9548,Z 129,A -71.7633,B 24.962,C -1.4224,E1 25.0592,E2 518.0582} C_DIS
LIN {X 43.2137,Y -115.0033,Z 129,A -73.1194,B 24.9622,C -1.4202,E1 25.0556,E2 519.4166} C_DIS
LIN {X 40.3783,Y -116.0292,Z 129,A -74.5626,B 24.9624,C -1.4166,E1 25.0518,E2 520.8656} C_DIS
LIN {X 37.1033,Y -117.1195,Z 129,A -76.1274,B 24.9624,C -1.4167,E1 25.0477,E2 522.427} C_DIS
LIN {X 34.6364,Y -117.8707,Z 129,A -77.327,B 24.9624,C -1.4155,E1 25.0444,E2 523.6274} C_DIS
LIN {X 31.7333,Y -118.6852,Z 129,A -78.7299,B 24.9625,C -1.4141,E1 25.0407,E2 525.0312} C_DIS
LIN {X 28.8111,Y -119.4282,Z 129,A -80.1743,B 24.9627,C -1.4109,E1 25.0367,E2 526.4813} C_DIS
LIN {X 25.8715,Y -120.0993,Z 129,A -81.5292,B 24.9627,C -1.412,E1 25.0331,E2 527.8316} C_DIS
LIN {X 22.4876,Y -120.7806,Z 129,A -83.1434,B 24.9627,C -1.4104,E1 25.0286,E2 529.4477} C_DIS
LIN {X 19.5167,Y -121.2961,Z 129,A -84.5475,B 24.9627,C -1.4094,E1 25.0248,E2 530.8527} C_DIS
LIN {X 16.5341,Y -121.7385,Z 129,A -85.9516,B 24.9628,C -1.4085,E1 25.0209,E2 532.2577} C_DIS
LIN {X 13.7708,Y -122.0808,Z 129,A -87.2333,B 24.9628,C -1.4085,E1 25.0173,E2 533.5384} C_DIS
LIN {X 10.9755,Y -122.363,Z 129,A -88.5983,B 24.963,C -1.4052,E1 25.0135,E2 534.9104} C_DIS
LIN {X 7.5336,Y -122.625,Z 129,A -90.1654,B 24.963,C -1.4065,E1 25.0092,E2 536.4737} C_DIS
LIN {X 4.522,Y -122.7729,Z 129,A -91.5706,B 24.963,C -1.406,E1 25.0052,E2 537.8797} C_DIS
LIN {X 1.5076,Y -122.8469,Z 129,A -92.9758,B 24.963,C -1.4057,E1 25.0013,E2 539.2856} C_DIS
LIN {X 1.5076,Y -122.8469,Z 129,A -92.9758,B 24.963,C -1.4057,E1 25.0013,E2 539.2856} C_DIS
Enddeposition()
LIN {X 0.8635,Y -121.9972,Z 129,A -92.7917,B 24.961,C -1.4436,E1 25.0021,E2 539.0116} C_DIS
Startdeposition()
$VEL.CP = VEL_PRINT
LIN {X 4.338,Y -121.9302,Z 129,A -91.0431,B 24.9606,C -1.4496,E1 25.007,E2 537.2491} C_DIS
LIN {X 8.1616,Y -121.7326,Z 129,A -89.3813,B 24.9609,C -1.4438,E1 25.0116,E2 535.6015} C_DIS
LIN {X 11.0174,Y -121.5076,Z 129,A -87.8729,B 24.9605,C -1.4523,E1 25.0158,E2 534.0739} C_DIS
LIN {X 14.0638,Y -121.1927,Z 129,A -86.1891,B 24.9598,C -1.465,E1 25.0206,E2 532.3612} C_DIS
LIN {X 19.2539,Y -120.4787,Z 129,A -83.7225,B 24.9597,C -1.4671,E1 25.0274,E2 529.8921} C_DIS
LIN {X 25.0366,Y -119.4105,Z 129,A -81.1315,B 24.96,C -1.4611,E1 25.0345,E2 527.3182} C_DIS
LIN {X 29.1225,Y -118.4794,Z 129,A -79.2713,B 24.9602,C -1.4579,E1 25.0395,E2 525.4684} C_DIS
LIN {X 32.8705,Y -117.4952,Z 129,A -77.3839,B 24.9599,C -1.4631,E1 25.0446,E2 523.5716} C_DIS
LIN {X 35.8747,Y -116.6127,Z 129,A -75.4797,B 24.9586,C -1.4861,E1 25.0498,E2 521.6164} C_DIS
LIN {X 39.7631,Y -115.3464,Z 129,A -74.0219,B 24.9598,C -1.4658,E1 25.0535,E2 520.2095} C_DIS
LIN {X 43.0178,Y -114.1707,Z 129,A -72.4122,B 24.9597,C -1.4673,E1 25.0578,E2 518.5997} C_DIS
LIN {X 46.2335,Y -112.9069,Z 129,A -70.7827,B 24.9595,C -1.4699,E1 25.062,E2 516.9676} C_DIS
LIN {X 51.5537,Y -110.5787,Z 129,A -68.1492,B 24.9595,C -1.4695,E1 25.0687,E2 514.3415} C_DIS
LIN {X 54.17,Y -109.3208,Z 129,A -66.7794,B 24.9595,C -1.4721,E1 25.0721,E2 512.9693} C_DIS
LIN {X 56.7242,Y -108.0177,Z 129,A -65.3279,B 24.959,C -1.4796,E1 25.0758,E2 511.5042} C_DIS
LIN {X 60.2408,Y -106.0984,Z 129,A -62.4274,B 24.9559,C -1.5338,E1 25.0831,E2 508.4841} C_DIS
LIN {X 66.0871,Y -102.5572,Z 129,A -60.3026,B 24.9586,C -1.4857,E1 25.0878,E2 506.4797} C_DIS
LIN {X 69.8336,Y -100.0438,Z 129,A -58.1231,B 24.9582,C -1.4931,E1 25.0929,E2 504.2903} C_DIS
LIN {X 72.8535,Y -97.8677,Z 129,A -56.3811,B 24.958,C -1.4965,E1 25.0968,E2 502.5465} C_DIS
LIN {X 75.874,Y -95.544,Z 129,A -54.6589,B 24.958,C -1.4971,E1 25.1006,E2 500.8292} C_DIS
LIN {X 79.6381,Y -92.432,Z 129,A -52.2813,B 24.9575,C -1.5065,E1 25.1057,E2 498.4386} C_DIS
LIN {X 82.5386,Y -89.8489,Z 129,A -50.5807,B 24.9575,C -1.5047,E1 25.1092,E2 496.7492} C_DIS
LIN {X 85.5067,Y -87.0295,Z 129,A -48.8749,B 24.9579,C -1.4985,E1 25.1126,E2 495.0649} C_DIS
LIN {X 87.5196,Y -85.0058,Z 129,A -47.2373,B 24.9569,C -1.5167,E1 25.1158,E2 493.3914} C_DIS
LIN {X 91.0164,Y -81.2495,Z 129,A -44.9337,B 24.9569,C -1.5176,E1 25.1202,E2 491.0959} C_DIS
LIN {X 93.6063,Y -78.2524,Z 129,A -43.1659,B 24.9569,C -1.5178,E1 25.1233,E2 489.3356} C_DIS
LIN {X 95.3899,Y -76.069,Z 129,A -41.6459,B 24.9561,C -1.5313,E1 25.126,E2 487.7909} C_DIS
LIN {X 98.3148,Y -72.2474,Z 129,A -39.6314,B 24.9564,C -1.5251,E1 25.1294,E2 485.8005} C_DIS
LIN {X 101.376,Y -67.8877,Z 129,A -37.0416,B 24.9558,C -1.5366,E1 25.1335,E2 483.1964} C_DIS
LIN {X 103.1714,Y -65.1263,Z 129,A -35.4469,B 24.9554,C -1.5435,E1 25.1359,E2 481.5935} C_DIS
LIN {X 104.8501,Y -62.386,Z 129,A -34.0999,B 24.9556,C -1.5397,E1 25.1379,E2 480.2623} C_DIS
LIN {X 106.4323,Y -59.6459,Z 129,A -32.4753,B 24.9549,C -1.5511,E1 25.1401,E2 478.6192} C_DIS
LIN {X 108.4182,Y -55.9568,Z 129,A -30.7125,B 24.9552,C -1.5467,E1 25.1424,E2 476.8762} C_DIS
LIN {X 109.6453,Y -53.5155,Z 129,A -29.2097,B 24.9543,C -1.5616,E1 25.1443,E2 475.3461} C_DIS
LIN {X 112.6039,Y -46.9682,Z 129,A -25.8594,B 24.9538,C -1.5708,E1 25.1481,E2 471.9925} C_DIS
LIN {X 114.6126,Y -41.8258,Z 129,A -23.2867,B 24.9533,C -1.578,E1 25.1506,E2 469.4172} C_DIS
LIN {X 116.0058,Y -37.7908,Z 129,A -21.4533,B 24.9535,C -1.5756,E1 25.1523,E2 467.5996} C_DIS
LIN {X 116.8119,Y -35.2236,Z 129,A -20.2555,B 24.9535,C -1.5763,E1 25.1532,E2 466.407} C_DIS
LIN {X 117.7396,Y -31.982,Z 129,A -18.5749,B 24.9528,C -1.5864,E1 25.1545,E2 464.7124} C_DIS
LIN {X 118.5594,Y -28.7946,Z 129,A -16.9599,B 24.9523,C -1.5949,E1 25.1556,E2 463.0867} C_DIS
LIN {X 119.4843,Y -24.6773,Z 129,A -15.3485,B 24.9531,C -1.5826,E1 25.1566,E2 461.5137} C_DIS
LIN {X 120.2911,Y -20.385,Z 129,A -12.9852,B 24.9517,C -1.605,E1 25.1578,E2 459.1113} C_DIS
LIN {X 120.8146,Y -17.0089,Z 129,A -11.43,B 24.9516,C -1.6078,E1 25.1584,E2 457.5588} C_DIS
LIN {X 121.307,Y -13.045,Z 129,A -9.7716,B 24.9519,C -1.6029,E1 25.1589,E2 455.9216} C_DIS
LIN {X 121.6812,Y -8.9224,Z 129,A -7.5139,B 24.9505,C -1.6251,E1 25.1595,E2 453.6249} C_DIS
LIN {X 121.8821,Y -5.4998,Z 129,A -6.247,B 24.9512,C -1.6131,E1 25.1596,E2 452.394} C_DIS
LIN {X 121.9948,Y -1.7264,Z 129,A -4.2109,B 24.9501,C -1.6322,E1 25.1598,E2 450.3249} C_DIS
LIN {X 121.9703,Y 3.0166,Z 129,A -1.782,B 24.949,C -1.6497,E1 25.1597,E2 447.8692} C_DIS
LIN {X 121.7479,Y 7.9351,Z 129,A 0.1582,B 24.9497,C -1.6384,E1 25.1594,E2 445.9672} C_DIS
LIN {X 121.5119,Y 10.9704,Z 129,A 1.5039,B 24.9497,C -1.6388,E1 25.1591,E2 444.6286} C_DIS
LIN {X 121.0488,Y 15.2576,Z 129,A 3.7914,B 24.9485,C -1.6586,E1 25.1583,E2 442.3079} C_DIS
LIN {X 120.0351,Y 21.8417,Z 129,A 6.6652,B 24.9486,C -1.6557,E1 25.1571,E2 439.4578} C_DIS
LIN {X 119.0645,Y 26.6366,Z 129,A 9.1923,B 24.9475,C -1.6745,E1 25.1556,E2 436.9011} C_DIS
LIN {X 118.3212,Y 29.7645,Z 129,A 10.6801,B 24.9472,C -1.6781,E1 25.1546,E2 435.4134} C_DIS
LIN {X 117.3839,Y 33.2636,Z 129,A 12.2217,B 24.9474,C -1.6754,E1 25.1535,E2 433.887} C_DIS
LIN {X 116.4185,Y 36.5008,Z 129,A 13.9148,B 24.9468,C -1.6856,E1 25.1521,E2 432.1795} C_DIS
LIN {X 115.2369,Y 40.0749,Z 129,A 15.625,B 24.9466,C -1.6881,E1 25.1505,E2 430.4731} C_DIS
LIN {X 113.9406,Y 43.6254,Z 129,A 17.4624,B 24.9461,C -1.6965,E1 25.1487,E2 428.6261} C_DIS
LIN {X 112.5021,Y 47.2097,Z 129,A 19.0649,B 24.9464,C -1.6913,E1 25.147,E2 427.0448} C_DIS
LIN {X 111.0538,Y 50.5241,Z 129,A 20.8847,B 24.9457,C -1.7023,E1 25.145,E2 425.209} C_DIS
LIN {X 109.4007,Y 54.0089,Z 129,A 22.5935,B 24.9457,C -1.7023,E1 25.1429,E2 423.5092} C_DIS
LIN {X 108.1321,Y 56.5069,Z 129,A 23.9049,B 24.9455,C -1.7058,E1 25.1412,E2 422.1966} C_DIS
LIN {X 106.8739,Y 58.855,Z 129,A 25.1351,B 24.9453,C -1.7082,E1 25.1396,E2 420.9671} C_DIS
LIN {X 103.4706,Y 64.6472,Z 129,A 28.3182,B 24.9447,C -1.7181,E1 25.135,E2 417.7769} C_DIS
LIN {X 100.6626,Y 68.9412,Z 129,A 30.8589,B 24.9439,C -1.7309,E1 25.131,E2 415.2187} C_DIS
LIN {X 98.1603,Y 72.4584,Z 129,A 32.7052,B 24.9441,C -1.7271,E1 25.128,E2 413.3903} C_DIS
LIN {X 95.8754,Y 75.4546,Z 129,A 34.4907,B 24.9438,C -1.7322,E1 25.125,E2 411.6011} C_DIS
LIN {X 93.879,Y 77.9241,Z 129,A 36.0205,B 24.9434,C -1.7377,E1 25.1223,E2 410.0655} C_DIS
LIN {X 91.1606,Y 81.0884,Z 129,A 37.9749,B 24.9431,C -1.742,E1 25.1187,E2 408.1096} C_DIS
LIN {X 88.3407,Y 84.1536,Z 129,A 39.9797,B 24.9427,C -1.7488,E1 25.1148,E2 406.0975} C_DIS
LIN {X 85.8586,Y 86.682,Z 129,A 41.613,B 24.9425,C -1.751,E1 25.1116,E2 404.4662} C_DIS
LIN {X 82.6133,Y 89.7804,Z 129,A 43.3816,B 24.9433,C -1.7388,E1 25.1081,E2 402.7336} C_DIS
LIN {X 80.6391,Y 91.5589,Z 129,A 44.9,B 24.9423,C -1.7545,E1 25.1049,E2 401.184} C_DIS
LIN {X 78.1138,Y 93.7214,Z 129,A 46.4304,B 24.9423,C -1.7561,E1 25.1016,E2 399.6559} C_DIS
LIN {X 75.4495,Y 95.8795,Z 129,A 48.0691,B 24.9419,C -1.7605,E1 25.098,E2 398.0129} C_DIS
LIN {X 72.1444,Y 98.3902,Z 129,A 49.9642,B 24.9419,C -1.7614,E1 25.0938,E2 396.1225} C_DIS
LIN {X 66.8625,Y 102.0538,Z 129,A 53.0888,B 24.9412,C -1.7715,E1 25.0866,E2 392.9844} C_DIS
LIN {X 62.8806,Y 104.5552,Z 129,A 55.1663,B 24.9414,C -1.7686,E1 25.0816,E2 390.9205} C_DIS
LIN {X 59.5883,Y 106.4645,Z 129,A 56.9241,B 24.9413,C -1.7698,E1 25.0774,E2 389.1652} C_DIS
LIN {X 57.3016,Y 107.7136,Z 129,A 58.1508,B 24.9412,C -1.7716,E1 25.0744,E2 387.9377} C_DIS
LIN {X 54.3294,Y 109.2418,Z 129,A 59.7351,B 24.941,C -1.7744,E1 25.0704,E2 386.3512} C_DIS
LIN {X 51.302,Y 110.6959,Z 129,A 61.3444,B 24.9408,C -1.7778,E1 25.0663,E2 384.7379} C_DIS
LIN {X 47.3183,Y 112.4563,Z 129,A 63.3808,B 24.9406,C -1.7797,E1 25.0611,E2 382.7019} C_DIS
LIN {X 44.0342,Y 113.784,Z 129,A 64.9813,B 24.9407,C -1.7783,E1 25.057,E2 381.1082} C_DIS
LIN {X 40.6683,Y 115.0287,Z 129,A 66.6984,B 24.9405,C -1.7814,E1 25.0525,E2 379.3873} C_DIS
LIN {X 37.9514,Y 115.9539,Z 129,A 68.0896,B 24.9403,C -1.7846,E1 25.0488,E2 377.9912} C_DIS
LIN {X 35.0495,Y 116.8636,Z 129,A 69.4611,B 24.9404,C -1.783,E1 25.0451,E2 376.6259} C_DIS
LIN {X 31.7223,Y 117.8098,Z 129,A 71.0966,B 24.9404,C -1.7847,E1 25.0407,E2 374.9892} C_DIS
LIN {X 27.951,Y 118.7621,Z 129,A 72.9188,B 24.9402,C -1.7855,E1 25.0358,E2 373.1677} C_DIS
LIN {X 21.3865,Y 120.117,Z 129,A 76.066,B 24.9402,C -1.7868,E1 25.0272,E2 370.0211} C_DIS
LIN {X 17.1343,Y 120.7967,Z 129,A 78.1606,B 24.9399,C -1.7909,E1 25.0214,E2 367.919} C_DIS
LIN {X 13.0047,Y 121.3112,Z 129,A 80.0505,B 24.9401,C -1.7882,E1 25.0161,E2 366.0368} C_DIS
LIN {X 9.5995,Y 121.6277,Z 129,A 81.4992,B 24.9406,C -1.781,E1 25.0122,E2 364.606} C_DIS
LIN {X 5.6631,Y 121.8751,Z 129,A 83.8638,B 24.9389,C -1.8049,E1 25.0054,E2 362.1855} C_DIS
LIN {X 2.3179,Y 121.9839,Z 129,A 85.0841,B 24.9401,C -1.7883,E1 25.0021,E2 361.0049} C_DIS
LIN {X -1.1012,Y 122.0014,Z 129,A 86.7015,B 24.9401,C -1.7885,E1 24.9976,E2 359.3871} C_DIS
LIN {X -7.101,Y 121.7996,Z 129,A 89.577,B 24.9399,C -1.7901,E1 24.9896,E2 356.507} C_DIS
LIN {X -13.6169,Y 121.245,Z 129,A 92.6444,B 24.9401,C -1.7884,E1 24.9811,E2 353.4422} C_DIS
LIN {X -17.1291,Y 120.7975,Z 129,A 94.0253,B 24.941,C -1.7744,E1 24.9773,E2 352.0933} C_DIS
LIN {X -22.4389,Y 119.9264,Z 129,A 96.8571,B 24.9402,C -1.7864,E1 24.9694,E2 349.2302} C_DIS
LIN {X -26.0131,Y 119.2005,Z 129,A 98.3781,B 24.9409,C -1.7762,E1 24.9653,E2 347.7317} C_DIS
LIN {X -28.8451,Y 118.547,Z 129,A 99.7746,B 24.9409,C -1.7764,E1 24.9615,E2 346.3329} C_DIS
LIN {X -33.0885,Y 117.4335,Z 129,A 101.9737,B 24.9406,C -1.7806,E1 24.9556,E2 344.1206} C_DIS
LIN {X -36.9805,Y 116.268,Z 129,A 104.0196,B 24.9403,C -1.7846,E1 24.9501,E2 342.0614} C_DIS
LIN {X -40.8178,Y 114.9763,Z 129,A 105.8363,B 24.9407,C -1.7784,E1 24.9453,E2 340.2561} C_DIS
LIN {X -43.9943,Y 113.7996,Z 129,A 107.3463,B 24.9411,C -1.7726,E1 24.9414,E2 338.7568} C_DIS
LIN {X -47.7344,Y 112.281,Z 129,A 109.2107,B 24.9414,C -1.7684,E1 24.9366,E2 336.8979} C_DIS
LIN {X -51.2311,Y 110.7289,Z 129,A 110.8971,B 24.9419,C -1.7608,E1 24.9323,E2 335.2257} C_DIS
LIN {X -53.4068,Y 109.6975,Z 129,A 112.1352,B 24.9417,C -1.7638,E1 24.9292,E2 333.9773} C_DIS
LIN {X -56.5413,Y 108.114,Z 129,A 113.8539,B 24.9417,C -1.7641,E1 24.9249,E2 332.253} C_DIS
LIN {X -63.4416,Y 104.2143,Z 129,A 117.7687,B 24.9415,C -1.766,E1 24.9154,E2 328.3221} C_DIS
LIN {X -67.2191,Y 101.8186,Z 129,A 119.659,B 24.9424,C -1.7525,E1 24.911,E2 326.4577} C_DIS
LIN {X -70.2032,Y 99.7869,Z 129,A 121.4591,B 24.9424,C -1.7537,E1 24.9069,E2 324.6487} C_DIS
LIN {X -73.1384,Y 97.6537,Z 129,A 123.1285,B 24.9427,C -1.7486,E1 24.9032,E2 322.9855} C_DIS
LIN {X -76.3621,Y 95.1557,Z 129,A 125.2037,B 24.9425,C -1.7516,E1 24.8986,E2 320.8956} C_DIS
LIN {X -79.7465,Y 92.3385,Z 129,A 127.0226,B 24.9435,C -1.7358,E1 24.8948,E2 319.1072} C_DIS
LIN {X -82.0094,Y 90.3345,Z 129,A 128.7275,B 24.9429,C -1.7452,E1 24.8912,E2 317.3732} C_DIS
LIN {X -85.0082,Y 87.5172,Z 129,A 130.5446,B 24.9436,C -1.7354,E1 24.8875,E2 315.5718} C_DIS
LIN {X -87.7469,Y 84.7699,Z 129,A 132.0822,B 24.9447,C -1.7184,E1 24.8846,E2 314.0681} C_DIS
LIN {X -89.8513,Y 82.536,Z 129,A 133.6085,B 24.9447,C -1.7185,E1 24.8817,E2 312.5349} C_DIS
LIN {X -91.4269,Y 80.7902,Z 129,A 134.8205,B 24.9445,C -1.7204,E1 24.8794,E2 311.3131} C_DIS
LIN {X -93.7266,Y 78.1076,Z 129,A 136.3827,B 24.9451,C -1.7118,E1 24.8766,E2 309.7641} C_DIS
LIN {X -95.6659,Y 75.7197,Z 129,A 138.1409,B 24.9444,C -1.7217,E1 24.8735,E2 307.9741} C_DIS
LIN {X -98.0085,Y 72.6658,Z 129,A 139.8176,B 24.9451,C -1.711,E1 24.8707,E2 306.315} C_DIS
LIN {X -100.2749,Y 69.5011,Z 129,A 141.6273,B 24.9455,C -1.7051,E1 24.8678,E2 304.5103} C_DIS
LIN {X -102.4164,Y 66.3064,Z 129,A 143.3587,B 24.9461,C -1.6967,E1 24.8651,E2 302.7903} C_DIS
LIN {X -104.2016,Y 63.4624,Z 129,A 145.0874,B 24.9459,C -1.6988,E1 24.8626,E2 301.0477} C_DIS
LIN {X -105.5598,Y 61.1783,Z 129,A 146.6087,B 24.9454,C -1.7071,E1 24.8604,E2 299.4987} C_DIS
LIN {X -107.891,Y 56.9647,Z 129,A 148.5581,B 24.9467,C -1.6867,E1 24.8579,E2 297.5875} C_DIS
LIN {X -109.3167,Y 54.1784,Z 129,A 150.0376,B 24.9469,C -1.6827,E1 24.856,E2 296.1096} C_DIS
LIN {X -110.5945,Y 51.5198,Z 129,A 151.635,B 24.9466,C -1.6878,E1 24.8541,E2 294.4915} C_DIS
LIN {X -112.2328,Y 47.8487,Z 129,A 153.3747,B 24.9474,C -1.6755,E1 24.8522,E2 292.7716} C_DIS
LIN {X -113.5061,Y 44.7416,Z 129,A 155.0371,B 24.9474,C -1.6743,E1 24.8505,E2 291.1027} C_DIS
LIN {X -114.8632,Y 41.1387,Z 129,A 156.9037,B 24.9477,C -1.6711,E1 24.8487,E2 289.2331} C_DIS
LIN {X -116.1381,Y 37.382,Z 129,A 158.6489,B 24.9484,C -1.6601,E1 24.8472,E2 287.5041} C_DIS
LIN {X -117.3224,Y 33.4805,Z 129,A 160.4659,B 24.949,C -1.6498,E1 24.8457,E2 285.7013} C_DIS
LIN {X -118.3357,Y 29.7081,Z 129,A 162.5172,B 24.9488,C -1.6533,E1 24.8443,E2 283.6297} C_DIS
LIN {X -119.1478,Y 26.2544,Z 129,A 163.9694,B 24.9497,C -1.6386,E1 24.8434,E2 282.2039} C_DIS
LIN {X -119.6823,Y 23.7065,Z 129,A 165.426,B 24.9493,C -1.6448,E1 24.8426,E2 280.724} C_DIS
LIN {X -120.4134,Y 19.654,Z 129,A 167.3846,B 24.9496,C -1.6396,E1 24.8416,E2 278.7662} C_DIS
LIN {X -120.9823,Y 15.7714,Z 129,A 169.025,B 24.9505,C -1.6248,E1 24.841,E2 277.1513} C_DIS
LIN {X -121.3362,Y 12.7662,Z 129,A 170.407,B 24.9509,C -1.6185,E1 24.8406,E2 275.7761} C_DIS
LIN {X -121.5873,Y 10.1052,Z 129,A 171.7742,B 24.9509,C -1.6192,E1 24.8403,E2 274.399} C_DIS
LIN {X -121.7793,Y 7.468,Z 129,A 173.1974,B 24.9506,C -1.623,E1 24.84,E2 272.9581} C_DIS
LIN {X -121.9609,Y 3.3388,Z 129,A 175.1505,B 24.951,C -1.6172,E1 24.8398,E2 271.007} C_DIS
LIN {X -122.0039,Y -0.7165,Z 129,A 176.8958,B 24.9518,C -1.604,E1 24.8398,E2 269.2826} C_DIS
LIN {X -121.9422,Y -3.9459,Z 129,A 178.4615,B 24.952,C -1.6012,E1 24.8399,E2 267.7142} C_DIS
LIN {X -121.7467,Y -7.9535,Z 129,A -179.6824,B 24.9524,C -1.5939,E1 24.8402,E2 265.8644} C_DIS
LIN {X -121.4938,Y -11.167,Z 129,A -178.1834,B 24.9527,C -1.5883,E1 24.8406,E2 264.3697} C_DIS
LIN {X -121.2342,Y -13.7091,Z 129,A -176.8776,B 24.9527,C -1.589,E1 24.841,E2 263.0544} C_DIS
LIN {X -120.7393,Y -17.5387,Z 129,A -174.9587,B 24.9527,C -1.5878,E1 24.8417,E2 261.1269} C_DIS
LIN {X -120.1643,Y -21.1235,Z 129,A -173.3731,B 24.9534,C -1.5772,E1 24.8424,E2 259.5572} C_DIS
LIN {X -119.5614,Y -24.3014,Z 129,A -171.848,B 24.9537,C -1.5726,E1 24.8432,E2 258.034} C_DIS
LIN {X -118.9802,Y -27.0068,Z 129,A -170.6239,B 24.9541,C -1.5653,E1 24.844,E2 256.8203} C_DIS
LIN {X -118.3748,Y -29.551,Z 129,A -169.3505,B 24.9542,C -1.5634,E1 24.8448,E2 255.5438} C_DIS
LIN {X -117.5729,Y -32.5951,Z 129,A -167.6708,B 24.954,C -1.5676,E1 24.8461,E2 253.8443} C_DIS
LIN {X -116.4749,Y -36.319,Z 129,A -165.9531,B 24.9546,C -1.5574,E1 24.8475,E2 252.141} C_DIS
LIN {X -115.2283,Y -40.0995,Z 129,A -164.1914,B 24.9552,C -1.547,E1 24.849,E2 250.394} C_DIS
LIN {X -113.7635,Y -44.0865,Z 129,A -162.2027,B 24.9555,C -1.5408,E1 24.851,E2 248.4089} C_DIS
LIN {X -112.6232,Y -46.9222,Z 129,A -160.5766,B 24.9553,C -1.545,E1 24.8527,E2 246.7639} C_DIS
LIN {X -111.2042,Y -50.1903,Z 129,A -158.9073,B 24.9556,C -1.54,E1 24.8546,E2 245.0973} C_DIS
LIN {X -109.4929,Y -53.8229,Z 129,A -157.0776,B 24.956,C -1.5321,E1 24.8568,E2 243.2764} C_DIS
LIN {X -108.2451,Y -56.2923,Z 129,A -155.6261,B 24.9558,C -1.5352,E1 24.8587,E2 241.8099} C_DIS
LIN {X -106.6833,Y -59.1965,Z 129,A -154.2032,B 24.9564,C -1.5253,E1 24.8605,E2 240.4029} C_DIS
LIN {X -105.2725,Y -61.6713,Z 129,A -152.8564,B 24.9566,C -1.5221,E1 24.8624,E2 239.0568} C_DIS
LIN {X -103.5521,Y -64.5168,Z 129,A -151.2896,B 24.9568,C -1.5182,E1 24.8647,E2 237.4914} C_DIS
LIN {X -101.9737,Y -66.984,Z 129,A -150.0586,B 24.9574,C -1.5082,E1 24.8666,E2 236.278} C_DIS
LIN {X -100.2557,Y -69.5288,Z 129,A -148.612,B 24.9576,C -1.5047,E1 24.8688,E2 234.8326} C_DIS
LIN {X -98.5083,Y -71.9831,Z 129,A -147.0743,B 24.9575,C -1.5065,E1 24.8714,E2 233.2829} C_DIS
LIN {X -95.7357,Y -75.6314,Z 129,A -144.925,B 24.9578,C -1.5011,E1 24.875,E2 231.1362} C_DIS
LIN {X -94.0402,Y -77.7302,Z 129,A -143.5638,B 24.9578,C -1.5023,E1 24.8774,E2 229.7659} C_DIS
LIN {X -91.2992,Y -80.9336,Z 129,A -141.4999,B 24.9578,C -1.5015,E1 24.8812,E2 227.6947} C_DIS
LIN {X -88.9331,Y -83.5245,Z 129,A -139.8866,B 24.9581,C -1.4962,E1 24.8843,E2 226.0868} C_DIS
LIN {X -86.2937,Y -86.2517,Z 129,A -138.0317,B 24.9581,C -1.4956,E1 24.8879,E2 224.2254} C_DIS
LIN {X -83.8673,Y -88.6108,Z 129,A -136.5079,B 24.9584,C -1.4893,E1 24.891,E2 222.7102} C_DIS
LIN {X -81.266,Y -91.0016,Z 129,A -134.9684,B 24.9589,C -1.4806,E1 24.8942,E2 221.1854} C_DIS
LIN {X -79.3728,Y -92.658,Z 129,A -133.7048,B 24.9589,C -1.482,E1 24.8968,E2 219.9135} C_DIS
LIN {X -76.8338,Y -94.7734,Z 129,A -132.2595,B 24.9593,C -1.4742,E1 24.8999,E2 218.4812} C_DIS
LIN {X -74.6838,Y -96.4772,Z 129,A -130.869,B 24.9592,C -1.4764,E1 24.903,E2 217.0803} C_DIS
LIN {X -68.5839,Y -100.9046,Z 129,A -127.2811,B 24.9594,C -1.4725,E1 24.9112,E2 213.4893} C_DIS
LIN {X -65.3825,Y -103.0095,Z 129,A -125.3603,B 24.9592,C -1.4752,E1 24.9157,E2 211.5559} C_DIS
LIN {X -62.1771,Y -104.9736,Z 129,A -123.7185,B 24.9597,C -1.4669,E1 24.9196,E2 209.9288} C_DIS
LIN {X -59.61,Y -106.4524,Z 129,A -122.3649,B 24.9599,C -1.4632,E1 24.9229,E2 208.58} C_DIS
LIN {X -56.8632,Y -107.9445,Z 129,A -120.855,B 24.9599,C -1.4632,E1 24.9266,E2 207.0659} C_DIS
LIN {X -53.5155,Y -109.6452,Z 129,A -118.9679,B 24.9597,C -1.4666,E1 24.9314,E2 205.1657} C_DIS
LIN {X -49.4806,Y -111.524,Z 129,A -116.9057,B 24.9599,C -1.463,E1 24.9366,E2 203.1071} C_DIS
LIN {X -45.8603,Y -113.0588,Z 129,A -115.0802,B 24.9601,C -1.4601,E1 24.9413,E2 201.2843} C_DIS
LIN {X -42.3464,Y -114.4227,Z 129,A -113.4737,B 24.9606,C -1.4508,E1 24.9454,E2 199.6965} C_DIS
LIN {X -39.6471,Y -115.3864,Z 129,A -111.8878,B 24.96,C -1.4608,E1 24.9497,E2 198.0838} C_DIS
LIN {X -36.1657,Y -116.5225,Z 129,A -110.3588,B 24.9606,C -1.4506,E1 24.9537,E2 196.5762} C_DIS
LIN {X -33.3559,Y -117.3577,Z 129,A -108.9899,B 24.9606,C -1.4493,E1 24.9574,E2 195.2082} C_DIS
LIN {X -29.6588,Y -118.3484,Z 129,A -106.5486,B 24.9591,C -1.4784,E1 24.9642,E2 192.6942} C_DIS
LIN {X -25.4854,Y -119.3156,Z 129,A -105.1289,B 24.9606,C -1.4496,E1 24.9679,E2 191.3413} C_DIS
LIN {X -21.1691,Y -120.1561,Z 129,A -102.9842,B 24.9605,C -1.4526,E1 24.9738,E2 189.1872} C_DIS
LIN {X -17.807,Y -120.7012,Z 129,A -101.297,B 24.9603,C -1.4563,E1 24.9785,E2 187.4898} C_DIS
LIN {X -14.0115,Y -121.1988,Z 129,A -99.6143,B 24.9606,C -1.4505,E1 24.9831,E2 185.8194} C_DIS
LIN {X -9.4445,Y -121.6401,Z 129,A -97.4418,B 24.9606,C -1.4512,E1 24.9891,E2 183.6442} C_DIS
LIN {X -5.9714,Y -121.8618,Z 129,A -95.6944,B 24.9602,C -1.4567,E1 24.9941,E2 181.8834} C_DIS
LIN {X -2.084,Y -121.9882,Z 129,A -93.9935,B 24.9606,C -1.451,E1 24.9988,E2 180.1958} C_DIS
LIN {X 0.8635,Y -121.9972,Z 129,A -92.7899,B 24.961,C -1.4428,E1 25.0021,E2 179.0116} C_DIS
Enddeposition()
LIN {X 0.8635,Y -121.9972,Z 129,A -92.7899,B 24.961,C -1.4428,E1 25.0021,E2 179.0116} C_DIS
Startdeposition()
$VEL.CP = VEL_PRINT
LIN {X 0.1647,Y -121.1592,Z 129,A -93.7332,B 24.9618,C -1.4286,E1 24.9994,E2 179.9886} C_DIS
LIN {X -3.7583,Y -121.0996,Z 129,A -95.5965,B 24.9618,C -1.428,E1 24.9941,E2 181.8536} C_DIS
LIN {X -7.8807,Y -120.9017,Z 129,A -97.9673,B 24.9628,C -1.4085,E1 24.9874,E2 184.2713} C_DIS
LIN {X -11.7722,Y -120.5863,Z 129,A -99.497,B 24.9621,C -1.4232,E1 24.9832,E2 185.7669} C_DIS
LIN {X -15.5699,Y -120.1533,Z 129,A -101.2981,B 24.9621,C -1.4238,E1 24.9782,E2 187.5677} C_DIS
LIN {X -19.781,Y -119.5324,Z 129,A -103.4031,B 24.9622,C -1.4202,E1 24.9724,E2 189.6833} C_DIS
LIN {X -23.4304,Y -118.8719,Z 129,A -105.1037,B 24.9621,C -1.4233,E1 24.9678,E2 191.3784} C_DIS
LIN {X -29.4753,Y -117.52,Z 129,A -107.97,B 24.9618,C -1.4276,E1 24.96,E2 194.2381} C_DIS
LIN {X -33.24,Y -116.5092,Z 129,A -109.7014,B 24.9615,C -1.434,E1 24.9554,E2 195.9572} C_DIS
LIN {X -36.5782,Y -115.5067,Z 129,A -111.598,B 24.962,C -1.4239,E1 24.9502,E2 197.8811} C_DIS
LIN {X -40.9534,Y -114.0281,Z 129,A -113.6251,B 24.9615,C -1.4329,E1 24.9449,E2 199.8907} C_DIS
LIN {X -44.427,Y -112.7187,Z 129,A -115.4884,B 24.9617,C -1.4297,E1 24.94,E2 201.7655} C_DIS
LIN {X -47.666,Y -111.3896,Z 129,A -117.2754,B 24.9619,C -1.4255,E1 24.9354,E2 203.5666} C_DIS
LIN {X -52.0764,Y -109.3959,Z 129,A -119.3236,B 24.9612,C -1.439,E1 24.9303,E2 205.5878} C_DIS
LIN {X -55.197,Y -107.8542,Z 129,A -120.8611,B 24.9608,C -1.446,E1 24.9265,E2 207.1129} C_DIS
LIN {X -57.7737,Y -106.4962,Z 129,A -122.2492,B 24.9608,C -1.4474,E1 24.9231,E2 208.5016} C_DIS
LIN {X -60.5506,Y -104.9424,Z 129,A -123.8384,B 24.9608,C -1.4457,E1 24.9192,E2 210.0994} C_DIS
LIN {X -64.0378,Y -102.8515,Z 129,A -125.7658,B 24.9607,C -1.4484,E1 24.9146,E2 212.0263} C_DIS
LIN {X -67.338,Y -100.7241,Z 129,A -127.864,B 24.9611,C -1.4406,E1 24.9096,E2 214.1499} C_DIS
LIN {X -72.9256,Y -96.753,Z 129,A -130.8167,B 24.9601,C -1.4591,E1 24.903,E2 217.0691} C_DIS
LIN {X -75.2299,Y -94.9722,Z 129,A -132.2523,B 24.9601,C -1.4591,E1 24.8999,E2 218.51} C_DIS
LIN {X -78.3874,Y -92.3835,Z 129,A -134.2027,B 24.96,C -1.4619,E1 24.8957,E2 220.4611} C_DIS
LIN {X -80.8749,Y -90.2135,Z 129,A -135.7815,B 24.9598,C -1.4642,E1 24.8924,E2 222.0407} C_DIS
LIN {X -83.9255,Y -87.383,Z 129,A -138.2094,B 24.9607,C -1.4482,E1 24.8874,E2 224.5167} C_DIS
LIN {X -86.7994,Y -84.531,Z 129,A -139.7331,B 24.9596,C -1.4694,E1 24.8845,E2 225.9965} C_DIS
LIN {X -91.8624,Y -78.999,Z 129,A -143.0877,B 24.9586,C -1.4858,E1 24.8782,E2 229.3269} C_DIS
LIN {X -93.8824,Y -76.5864,Z 129,A -144.76,B 24.9589,C -1.4813,E1 24.8752,E2 231.0175} C_DIS
LIN {X -97.2168,Y -72.3082,Z 129,A -147.4159,B 24.9588,C -1.4837,E1 24.8707,E2 233.6806} C_DIS
LIN {X -99.4995,Y -69.131,Z 129,A -149.1033,B 24.9581,C -1.4955,E1 24.868,E2 235.3481} C_DIS
LIN {X -101.5916,Y -66.0214,Z 129,A -150.8531,B 24.9578,C -1.501,E1 24.8653,E2 237.0935} C_DIS
LIN {X -103.7712,Y -62.5377,Z 129,A -153.1909,B 24.9585,C -1.4892,E1 24.8618,E2 239.4714} C_DIS
LIN {X -105.3979,Y -59.7579,Z 129,A -154.3665,B 24.9574,C -1.5083,E1 24.8603,E2 240.6076} C_DIS
LIN {X -106.9113,Y -57.0053,Z 129,A -155.8946,B 24.9573,C -1.5106,E1 24.8582,E2 242.1384} C_DIS
LIN {X -108.4612,Y -53.9948,Z 129,A -157.5216,B 24.9571,C -1.514,E1 24.8562,E2 243.766} C_DIS
LIN {X -109.8981,Y -51.0066,Z 129,A -159.1139,B 24.9569,C -1.5174,E1 24.8543,E2 245.3587} C_DIS
LIN {X -111.1679,Y -48.1768,Z 129,A -160.5386,B 24.9565,C -1.5235,E1 24.8527,E2 246.7769} C_DIS
LIN {X -112.3628,Y -45.3208,Z 129,A -162.0271,B 24.9563,C -1.5267,E1 24.8511,E2 248.2659} C_DIS
LIN {X -114.4877,Y -39.649,Z 129,A -164.8155,B 24.9557,C -1.5385,E1 24.8484,E2 251.0419} C_DIS
LIN {X -115.3342,Y -37.112,Z 129,A -166.2527,B 24.9559,C -1.535,E1 24.8472,E2 252.4958} C_DIS
LIN {X -117.1465,Y -30.9246,Z 129,A -169.4127,B 24.9556,C -1.5396,E1 24.8447,E2 255.663} C_DIS
LIN {X -117.981,Y -27.5648,Z 129,A -170.9342,B 24.955,C -1.5497,E1 24.8438,E2 257.1694} C_DIS
LIN {X -118.7725,Y -23.9278,Z 129,A -172.6567,B 24.9546,C -1.5569,E1 24.8428,E2 258.8851} C_DIS
LIN {X -119.4439,Y -20.3099,Z 129,A -174.4747,B 24.9545,C -1.5591,E1 24.8419,E2 260.7085} C_DIS
LIN {X -119.9521,Y -17.0507,Z 129,A -176.0047,B 24.9541,C -1.5653,E1 24.8412,E2 262.2327} C_DIS
LIN {X -120.3608,Y -13.8768,Z 129,A -177.5144,B 24.9538,C -1.5704,E1 24.8407,E2 263.7395} C_DIS
LIN {X -120.7268,Y -10.2279,Z 129,A -179.3394,B 24.9537,C -1.5721,E1 24.8403,E2 265.5714} C_DIS
LIN {X -120.97,Y -6.7444,Z 129,A 179.0793,B 24.9532,C -1.5805,E1 24.84,E2 267.1422} C_DIS
LIN {X -121.1115,Y -3.3699,Z 129,A 177.4833,B 24.9529,C -1.5857,E1 24.8398,E2 268.7353} C_DIS
LIN {X -121.1581,Y 0.3814,Z 129,A 175.6076,B 24.9528,C -1.5872,E1 24.8398,E2 270.6188} C_DIS
LIN {X -121.0957,Y 3.8856,Z 129,A 174.0232,B 24.9523,C -1.5957,E1 24.8399,E2 272.1924} C_DIS
LIN {X -120.964,Y 6.8528,Z 129,A 172.5955,B 24.9521,C -1.5993,E1 24.8401,E2 273.6201} C_DIS
LIN {X -120.7218,Y 10.29,Z 129,A 170.813,B 24.9521,C -1.5981,E1 24.8405,E2 275.4161} C_DIS
LIN {X -120.331,Y 14.1309,Z 129,A 169.1266,B 24.9514,C -1.6101,E1 24.841,E2 277.0842} C_DIS
LIN {X -119.9258,Y 17.2358,Z 129,A 167.6364,B 24.9512,C -1.6145,E1 24.8416,E2 278.5727} C_DIS
LIN {X -119.4579,Y 20.2263,Z 129,A 166.2098,B 24.9509,C -1.6193,E1 24.8422,E2 279.9962} C_DIS
LIN {X -118.8691,Y 23.4449,Z 129,A 164.588,B 24.9508,C -1.6212,E1 24.843,E2 281.6231} C_DIS
LIN {X -118.0611,Y 27.2181,Z 129,A 162.7688,B 24.9504,C -1.6274,E1 24.8441,E2 283.4384} C_DIS
LIN {X -116.3869,Y 33.6714,Z 129,A 159.4544,B 24.9502,C -1.6306,E1 24.8466,E2 286.7645} C_DIS
LIN {X -115.2802,Y 37.2787,Z 129,A 157.7637,B 24.9496,C -1.6403,E1 24.848,E2 288.4418} C_DIS
LIN {X -113.1073,Y 43.4313,Z 129,A 154.6421,B 24.9491,C -1.6484,E1 24.8509,E2 291.5616} C_DIS
LIN {X -111.6859,Y 46.9628,Z 129,A 152.8852,B 24.9486,C -1.6558,E1 24.8528,E2 293.3106} C_DIS
LIN {X -108.7851,Y 53.3414,Z 129,A 149.676,B 24.9477,C -1.6703,E1 24.8565,E2 296.5027} C_DIS
LIN {X -107.3096,Y 56.249,Z 129,A 147.078,B 24.9502,C -1.6303,E1 24.86,E2 299.2099} C_DIS
LIN {X -104.4336,Y 61.4241,Z 129,A 145.3702,B 24.9468,C -1.6847,E1 24.8622,E2 300.797} C_DIS
LIN {X -102.7824,Y 64.1484,Z 129,A 143.6477,B 24.9471,C -1.6798,E1 24.8648,E2 302.54} C_DIS
LIN {X -100.7725,Y 67.2653,Z 129,A 141.5694,B 24.9477,C -1.671,E1 24.868,E2 304.6499} C_DIS
LIN {X -98.415,Y 70.6672,Z 129,A 139.9455,B 24.9464,C -1.6906,E1 24.8706,E2 306.2349} C_DIS
LIN {X -95.3693,Y 74.7274,Z 129,A 137.6503,B 24.9457,C -1.7017,E1 24.8744,E2 308.5147} C_DIS
LIN {X -92.6599,Y 78.0629,Z 129,A 135.3538,B 24.9461,C -1.6957,E1 24.8785,E2 310.8361} C_DIS
LIN {X -90.258,Y 80.8253,Z 129,A 133.7244,B 24.9455,C -1.7046,E1 24.8815,E2 312.4517} C_DIS
LIN {X -87.8108,Y 83.4801,Z 129,A 132.0527,B 24.9452,C -1.7104,E1 24.8847,E2 314.1169} C_DIS
LIN {X -85.0054,Y 86.3328,Z 129,A 130.0711,B 24.9452,C -1.7112,E1 24.8886,E2 316.1049} C_DIS
LIN {X -81.6843,Y 89.4818,Z 129,A 127.8151,B 24.945,C -1.7124,E1 24.8932,E2 318.3673} C_DIS
LIN {X -78.64,Y 92.1683,Z 129,A 126.0273,B 24.9444,C -1.7225,E1 24.897,E2 320.138} C_DIS
LIN {X -74.9199,Y 95.2172,Z 129,A 123.7683,B 24.944,C -1.7282,E1 24.9019,E2 322.3921} C_DIS
LIN {X -72.5866,Y 97.0076,Z 129,A 122.3123,B 24.944,C -1.7283,E1 24.9051,E2 323.853} C_DIS
LIN {X -68.9389,Y 99.633,Z 129,A 120.2159,B 24.9437,C -1.7339,E1 24.9099,E2 325.9433} C_DIS
LIN {X -65.8491,Y 101.7023,Z 129,A 118.2381,B 24.9441,C -1.7278,E1 24.9145,E2 327.942} C_DIS
LIN {X -61.3894,Y 104.4541,Z 129,A 115.378,B 24.9448,C -1.7158,E1 24.9215,E2 330.8394} C_DIS
LIN {X -57.7147,Y 106.5282,Z 129,A 114.2139,B 24.9422,C -1.7556,E1 24.9241,E2 331.9122} C_DIS
LIN {X -55.2654,Y 107.8193,Z 129,A 112.5618,B 24.9431,C -1.7428,E1 24.9283,E2 333.5994} C_DIS
LIN {X -52.0427,Y 109.4122,Z 129,A 110.7892,B 24.9431,C -1.7423,E1 24.9327,E2 335.3778} C_DIS
LIN {X -48.6144,Y 110.9771,Z 129,A 109.1115,B 24.9426,C -1.7496,E1 24.937,E2 337.0421} C_DIS
LIN {X -43.5751,Y 113.0529,Z 129,A 106.5841,B 24.9422,C -1.7554,E1 24.9435,E2 339.5613} C_DIS
LIN {X -40.7472,Y 114.1023,Z 129,A 104.9454,B 24.9427,C -1.7478,E1 24.9479,E2 341.2212} C_DIS
LIN {X -36.8576,Y 115.4165,Z 129,A 103.1213,B 24.9422,C -1.7554,E1 24.9526,E2 343.0308} C_DIS
LIN {X -33.1687,Y 116.5294,Z 129,A 101.3161,B 24.9421,C -1.7582,E1 24.9575,E2 344.8323} C_DIS
LIN {X -30.1599,Y 117.344,Z 129,A 99.8369,B 24.942,C -1.7595,E1 24.9615,E2 346.3107} C_DIS
LIN {X -26.6711,Y 118.1874,Z 129,A 98.0316,B 24.9422,C -1.7562,E1 24.9664,E2 348.1261} C_DIS
LIN {X -22.8224,Y 118.989,Z 129,A 95.6173,B 24.9437,C -1.7331,E1 24.9732,E2 350.5981} C_DIS
LIN {X -18.0393,Y 119.8084,Z 129,A 94.0469,B 24.9415,C -1.767,E1 24.9773,E2 352.0894} C_DIS
LIN {X -9.5239,Y 120.7831,Z 129,A 88.9399,B 24.9444,C -1.722,E1 24.9918,E2 357.3059} C_DIS
LIN {X -3.1849,Y 121.1172,Z 129,A 87.4034,B 24.94,C -1.789,E1 24.9957,E2 358.6838} C_DIS
LIN {X 2.4513,Y 121.1333,Z 129,A 84.5347,B 24.9406,C -1.7802,E1 25.0037,E2 361.5734} C_DIS
LIN {X 8.2312,Y 120.878,Z 129,A 81.8025,B 24.9406,C -1.7804,E1 25.0113,E2 364.3042} C_DIS
LIN {X 14.6407,Y 120.2713,Z 129,A 78.6344,B 24.941,C -1.7743,E1 25.0202,E2 367.4849} C_DIS
LIN {X 18.8052,Y 119.69,Z 129,A 76.4834,B 24.9415,C -1.7662,E1 25.0262,E2 369.653} C_DIS
LIN {X 23.2977,Y 118.8975,Z 129,A 74.0456,B 24.9424,C -1.7524,E1 25.0329,E2 372.1207} C_DIS
LIN {X 28.4051,Y 117.7815,Z 129,A 71.8093,B 24.9418,C -1.762,E1 25.0389,E2 374.3312} C_DIS
LIN {X 32.1659,Y 116.8115,Z 129,A 69.9617,B 24.9419,C -1.7603,E1 25.0439,E2 376.18} C_DIS
LIN {X 36.15,Y 115.6395,Z 129,A 68.0443,B 24.9419,C -1.761,E1 25.049,E2 378.0924} C_DIS
LIN {X 39.9477,Y 114.3829,Z 129,A 66.1677,B 24.9419,C -1.7601,E1 25.054,E2 379.9675} C_DIS
LIN {X 43.8531,Y 112.9441,Z 129,A 64.3057,B 24.9417,C -1.7631,E1 25.0588,E2 381.8183} C_DIS
LIN {X 47.5912,Y 111.4211,Z 129,A 62.3557,B 24.942,C -1.7591,E1 25.0639,E2 383.7732} C_DIS
LIN {X 50.8662,Y 109.9634,Z 129,A 60.6088,B 24.9423,C -1.7547,E1 25.0683,E2 385.5261} C_DIS
LIN {X 54.0252,Y 108.4462,Z 129,A 58.8802,B 24.9426,C -1.7493,E1 25.0727,E2 387.263} C_DIS
LIN {X 57.7023,Y 106.5349,Z 129,A 56.9765,B 24.9426,C -1.7493,E1 25.0774,E2 389.1613} C_DIS
LIN {X 61.2857,Y 104.5154,Z 129,A 54.9149,B 24.9432,C -1.7409,E1 25.0824,E2 391.2365} C_DIS
LIN {X 64.8037,Y 102.3731,Z 129,A 52.9455,B 24.9435,C -1.7369,E1 25.0871,E2 393.2093} C_DIS
LIN {X 70.3475,Y 98.6432,Z 129,A 50.0553,B 24.943,C -1.7444,E1 25.0937,E2 396.0719} C_DIS
LIN {X 72.9038,Y 96.7693,Z 129,A 48.4669,B 24.9434,C -1.7374,E1 25.0973,E2 397.671} C_DIS
LIN {X 76.1603,Y 94.2277,Z 129,A 46.5597,B 24.9435,C -1.736,E1 25.1014,E2 399.5745} C_DIS
LIN {X 78.6991,Y 92.1179,Z 129,A 45.018,B 24.9437,C -1.7339,E1 25.1047,E2 401.1153} C_DIS
LIN {X 82.6296,Y 88.6106,Z 129,A 42.6503,B 24.9437,C -1.7347,E1 25.1096,E2 403.4716} C_DIS
LIN {X 85.4639,Y 85.8799,Z 129,A 40.5636,B 24.9446,C -1.7199,E1 25.1138,E2 405.5846} C_DIS
LIN {X 88.0804,Y 83.1935,Z 129,A 38.8115,B 24.9448,C -1.717,E1 25.1172,E2 407.3359} C_DIS
LIN {X 90.3698,Y 80.7004,Z 129,A 37.334,B 24.9446,C -1.7193,E1 25.12,E2 408.8014} C_DIS
LIN {X 92.6262,Y 78.1025,Z 129,A 35.5614,B 24.9453,C -1.7084,E1 25.1232,E2 410.5917} C_DIS
LIN {X 95.1989,Y 74.943,Z 129,A 33.8359,B 24.945,C -1.7135,E1 25.1262,E2 412.2971} C_DIS
LIN {X 97.0362,Y 72.5486,Z 129,A 32.3171,B 24.9455,C -1.7055,E1 25.1288,E2 413.8275} C_DIS
LIN {X 99.4029,Y 69.2699,Z 129,A 30.1473,B 24.9466,C -1.6881,E1 25.1323,E2 416.0278} C_DIS
LIN {X 102.0209,Y 65.3528,Z 129,A 28.1084,B 24.9464,C -1.6914,E1 25.1354,E2 418.0485} C_DIS
LIN {X 105.6719,Y 59.2683,Z 129,A 25.1503,B 24.9457,C -1.7018,E1 25.1396,E2 420.9671} C_DIS
LIN {X 107.4134,Y 56.0517,Z 129,A 23.0417,B 24.9472,C -1.6784,E1 25.1424,E2 423.1199} C_DIS
LIN {X 109.2186,Y 52.4456,Z 129,A 21.2752,B 24.9472,C -1.6798,E1 25.1446,E2 424.8734} C_DIS
LIN {X 110.5953,Y 49.4774,Z 129,A 19.4322,B 24.9483,C -1.6609,E1 25.1467,E2 426.7512} C_DIS
LIN {X 112.5524,Y 44.8502,Z 129,A 16.9264,B 24.9491,C -1.6475,E1 25.1494,E2 429.2747} C_DIS
LIN {X 113.8729,Y 41.3791,Z 129,A 15.9494,B 24.9471,C -1.6805,E1 25.1503,E2 430.1683} C_DIS
LIN {X 114.7675,Y 38.8289,Z 129,A 14.3834,B 24.9482,C -1.6624,E1 25.1517,E2 431.7682} C_DIS
LIN {X 115.7876,Y 35.6724,Z 129,A 12.8371,B 24.9484,C -1.6587,E1 25.153,E2 433.3144} C_DIS
LIN {X 116.7728,Y 32.3092,Z 129,A 11.0312,B 24.9492,C -1.6462,E1 25.1544,E2 435.1394} C_DIS
LIN {X 117.7377,Y 28.5847,Z 129,A 9.3568,B 24.9492,C -1.6477,E1 25.1555,E2 436.8006} C_DIS
LIN {X 118.6162,Y 24.6888,Z 129,A 7.6329,B 24.949,C -1.6499,E1 25.1566,E2 438.5093} C_DIS
LIN {X 119.148,Y 21.9839,Z 129,A 5.4437,B 24.9519,C -1.6022,E1 25.1577,E2 440.7982} C_DIS
LIN {X 119.9649,Y 16.9609,Z 129,A 3.4829,B 24.951,C -1.6163,E1 25.1585,E2 442.7141} C_DIS
LIN {X 120.642,Y 11.1693,Z 129,A 1.2146,B 24.9501,C -1.6316,E1 25.1592,E2 444.933} C_DIS
LIN {X 121.0738,Y 4.5598,Z 129,A -2.8278,B 24.9534,C -1.5765,E1 25.1598,E2 449.0813} C_DIS
LIN {X 121.1563,Y -0.6646,Z 129,A -5.3792,B 24.9541,C -1.5645,E1 25.1598,E2 451.6458} C_DIS
LIN {X 120.9879,Y -6.4215,Z 129,A -7.1194,B 24.9518,C -1.604,E1 25.1595,E2 453.2825} C_DIS
LIN {X 120.4095,Y -13.4606,Z 129,A -10.4977,B 24.9526,C -1.5911,E1 25.1587,E2 456.6713} C_DIS
LIN {X 119.4557,Y -20.2397,Z 129,A -13.9861,B 24.9539,C -1.568,E1 25.1573,E2 460.1934} C_DIS
LIN {X 118.6404,Y -24.5711,Z 129,A -15.793,B 24.9535,C -1.575,E1 25.1563,E2 461.9734} C_DIS
LIN {X 117.9576,Y -27.6661,Z 129,A -17.4326,B 24.9542,C -1.5632,E1 25.1553,E2 463.6314} C_DIS
LIN {X 116.9365,Y -31.7035,Z 129,A -19.2242,B 24.9541,C -1.5657,E1 25.154,E2 465.4068} C_DIS
LIN {X 116.0578,Y -34.784,Z 129,A -20.7237,B 24.9543,C -1.5616,E1 25.1528,E2 466.9074} C_DIS
LIN {X 115.1943,Y -37.5442,Z 129,A -22.08,B 24.9545,C -1.5578,E1 25.1517,E2 468.2649} C_DIS
LIN {X 114.217,Y -40.4206,Z 129,A -23.8245,B 24.9557,C -1.538,E1 25.15,E2 470.0464} C_DIS
LIN {X 112.8162,Y -44.1786,Z 129,A -25.4345,B 24.9552,C -1.5462,E1 25.1485,E2 471.6279} C_DIS
LIN {X 111.391,Y -47.6626,Z 129,A -27.8769,B 24.9574,C -1.508,E1 25.1457,E2 474.147} C_DIS
LIN {X 109.4208,Y -52.0248,Z 129,A -29.3144,B 24.9555,C -1.5418,E1 25.1441,E2 475.497} C_DIS
LIN {X 107.6222,Y -55.6509,Z 129,A -31.3753,B 24.9562,C -1.5287,E1 25.1415,E2 477.5778} C_DIS
LIN {X 105.1064,Y -60.2652,Z 129,A -33.8417,B 24.9566,C -1.5223,E1 25.1382,E2 480.0465} C_DIS
LIN {X 103.3671,Y -63.2028,Z 129,A -35.6651,B 24.9574,C -1.5072,E1 25.1355,E2 481.8961} C_DIS
LIN {X 101.0899,Y -66.7839,Z 129,A -37.447,B 24.9571,C -1.5126,E1 25.1328,E2 483.6565} C_DIS
LIN {X 98.3665,Y -70.7352,Z 129,A -40.5467,B 24.9598,C -1.4656,E1 25.1277,E2 486.8519} C_DIS
LIN {X 94.9224,Y -75.2929,Z 129,A -42.4185,B 24.9579,C -1.4987,E1 25.1246,E2 488.6367} C_DIS
LIN {X 90.4453,Y -80.6161,Z 129,A -45.6608,B 24.9583,C -1.4923,E1 25.1187,E2 491.8793} C_DIS
LIN {X 86.3552,Y -84.9827,Z 129,A -48.1984,B 24.9579,C -1.4995,E1 25.1139,E2 494.3889} C_DIS
LIN {X 83.2955,Y -87.9845,Z 129,A -50.5808,B 24.9591,C -1.4771,E1 25.109,E2 496.8143} C_DIS
LIN {X 80.1884,Y -90.8267,Z 129,A -53.1013,B 24.9608,C -1.4467,E1 25.1037,E2 499.3965} C_DIS
LIN {X 76.625,Y -93.8511,Z 129,A -54.7027,B 24.9595,C -1.4712,E1 25.1003,E2 500.9339} C_DIS
LIN {X 74,Y -95.9336,Z 129,A -56.4897,B 24.9602,C -1.4579,E1 25.0963,E2 502.7458} C_DIS
LIN {X 68.0584,Y -100.2363,Z 129,A -59.6934,B 24.9599,C -1.4636,E1 25.0891,E2 505.925} C_DIS
LIN {X 64.147,Y -102.7833,Z 129,A -62.4784,B 24.9616,C -1.4314,E1 25.0824,E2 508.777} C_DIS
LIN {X 60.3076,Y -105.082,Z 129,A -64.0025,B 24.9603,C -1.456,E1 25.0789,E2 510.2384} C_DIS
LIN {X 56.4821,Y -107.1868,Z 129,A -66.0382,B 24.9604,C -1.4537,E1 25.0739,E2 512.2735} C_DIS
LIN {X 53.6191,Y -108.6474,Z 129,A -67.582,B 24.9606,C -1.45,E1 25.07,E2 513.8219} C_DIS
LIN {X 45.2662,Y -112.3851,Z 129,A -71.7283,B 24.9606,C -1.4521,E1 25.0595,E2 517.9533} C_DIS
LIN {X 40.1618,Y -114.3078,Z 129,A -75.0546,B 24.9626,C -1.413,E1 25.0505,E2 521.3649} C_DIS
LIN {X 35.8725,Y -115.7255,Z 129,A -76.5573,B 24.9611,C -1.4405,E1 25.0467,E2 522.7999} C_DIS
LIN {X 32.5958,Y -116.6917,Z 129,A -78.1683,B 24.9612,C -1.4389,E1 25.0423,E2 524.4121} C_DIS
LIN {X 28.9579,Y -117.6467,Z 129,A -79.9936,B 24.9614,C -1.4348,E1 25.0374,E2 526.2441} C_DIS
LIN {X 25.8854,Y -118.3604,Z 129,A -81.4504,B 24.9614,C -1.4351,E1 25.0334,E2 527.6984} C_DIS
LIN {X 19.0012,Y -119.6597,Z 129,A -84.6179,B 24.9612,C -1.4392,E1 25.0248,E2 530.8526} C_DIS
LIN {X 13.5223,Y -120.4023,Z 129,A -87.3235,B 24.9615,C -1.4331,E1 25.0173,E2 533.5703} C_DIS
LIN {X 10.3894,Y -120.7139,Z 129,A -89.4376,B 24.9631,C -1.4031,E1 25.0112,E2 535.7543} C_DIS
LIN {X 6.0544,Y -121.0082,Z 129,A -90.8793,B 24.9616,C -1.4308,E1 25.0073,E2 537.1298} C_DIS
LIN {X 0.8474,Y -121.1463,Z 129,A -92.4071,B 24.9593,C -1.4743,E1 25.0034,E2 538.5543} C_DIS
Enddeposition()
LIN {X 0.8474,Y -121.1463,Z 129,A -92.4071,B 24.9593,C -1.4743,E1 25.0034,E2 538.5543} C_DIS
Startdeposition()
$VEL.CP = VEL_PRINT
LIN {X 6.1362,Y -120.1544,Z 129,A -89.0702,B 24.9562,C -1.5287,E1 25.013,E2 535.0897} C_DIS
LIN {X 12.9262,Y -119.6142,Z 129,A -87.3359,B 24.9601,C -1.4586,E1 25.0174,E2 533.5225} C_DIS
LIN {X 18.463,Y -118.8848,Z 129,A -84.308,B 24.9591,C -1.4776,E1 25.0259,E2 530.452} C_DIS
LIN {X 24.0262,Y -117.8866,Z 129,A -81.602,B 24.9589,C -1.4805,E1 25.0333,E2 527.7422} C_DIS
LIN {X 27.5338,Y -117.1178,Z 129,A -79.82,B 24.9587,C -1.4856,E1 25.0382,E2 525.9506} C_DIS
LIN {X 31.2584,Y -116.1783,Z 129,A -78.1482,B 24.959,C -1.48,E1 25.0427,E2 524.2947} C_DIS
LIN {X 34.24,Y -115.3347,Z 129,A -76.6353,B 24.9588,C -1.4834,E1 25.0467,E2 522.7761} C_DIS
LIN {X 36.5479,Y -114.6254,Z 129,A -74.2715,B 24.9554,C -1.5436,E1 25.0534,E2 520.2745} C_DIS
LIN {X 43.3099,Y -112.2464,Z 129,A -71.9331,B 24.9581,C -1.4959,E1 25.0592,E2 518.054} C_DIS
LIN {X 46.5637,Y -110.9339,Z 129,A -69.5233,B 24.9559,C -1.5343,E1 25.0656,E2 515.559} C_DIS
LIN {X 51.7217,Y -108.6256,Z 129,A -67.6033,B 24.9578,C -1.501,E1 25.0702,E2 513.7227} C_DIS
LIN {X 55.4386,Y -106.7779,Z 129,A -65.7712,B 24.958,C -1.4973,E1 25.0748,E2 511.9044} C_DIS
LIN {X 59.8726,Y -104.354,Z 129,A -63.6403,B 24.9585,C -1.4882,E1 25.0799,E2 509.801} C_DIS
LIN {X 62.1472,Y -103.0163,Z 129,A -61.453,B 24.9558,C -1.536,E1 25.0854,E2 507.5077} C_DIS
LIN {X 65.9796,Y -100.6044,Z 129,A -59.9235,B 24.9573,C -1.5095,E1 25.0888,E2 506.0458} C_DIS
LIN {X 68.7032,Y -98.7641,Z 129,A -58.0395,B 24.9562,C -1.5283,E1 25.0932,E2 504.1238} C_DIS
LIN {X 75.393,Y -93.7581,Z 129,A -54.3427,B 24.9565,C -1.523,E1 25.1014,E2 500.453} C_DIS
LIN {X 80.7046,Y -89.2279,Z 129,A -51.0396,B 24.9562,C -1.5296,E1 25.1084,E2 497.1473} C_DIS
LIN {X 85.1862,Y -84.9595,Z 129,A -47.9848,B 24.9554,C -1.5421,E1 25.1145,E2 494.0759} C_DIS
LIN {X 89.4931,Y -80.4083,Z 129,A -44.4169,B 24.9533,C -1.5788,E1 25.1214,E2 490.437} C_DIS
LIN {X 93.0013,Y -76.3267,Z 129,A -42.5458,B 24.9549,C -1.5511,E1 25.1246,E2 488.6399} C_DIS
LIN {X 98.2816,Y -69.3942,Z 129,A -38.3913,B 24.9542,C -1.5627,E1 25.1315,E2 484.4779} C_DIS
LIN {X 100.5141,Y -66.1166,Z 129,A -36.6274,B 24.9542,C -1.5619,E1 25.1343,E2 482.7247} C_DIS
LIN {X 103.7015,Y -60.9963,Z 129,A -34.1102,B 24.9548,C -1.5526,E1 25.1379,E2 480.2422} C_DIS
LIN {X 106.1535,Y -56.6243,Z 129,A -31.3963,B 24.9535,C -1.5758,E1 25.1416,E2 477.4877} C_DIS
LIN {X 107.7324,Y -53.5558,Z 129,A -29.7927,B 24.9533,C -1.5788,E1 25.1436,E2 475.8855} C_DIS
LIN {X 110.4938,Y -47.601,Z 129,A -26.5636,B 24.9524,C -1.5935,E1 25.1474,E2 472.6393} C_DIS
LIN {X 111.9724,Y -44.0074,Z 129,A -24.8328,B 24.9524,C -1.5933,E1 25.1492,E2 470.9185} C_DIS
LIN {X 113.7438,Y -39.208,Z 129,A -22.2516,B 24.9515,C -1.6082,E1 25.1516,E2 468.3167} C_DIS
LIN {X 114.9032,Y -35.6613,Z 129,A -20.6571,B 24.9517,C -1.6048,E1 25.153,E2 466.7393} C_DIS
LIN {X 115.8611,Y -32.4166,Z 129,A -18.9912,B 24.9513,C -1.6127,E1 25.1543,E2 465.0643} C_DIS
LIN {X 116.7914,Y -28.8856,Z 129,A -17.2964,B 24.9511,C -1.6161,E1 25.1554,E2 463.3712} C_DIS
Enddeposition()
END
